LIN {X 0,Y 523.426,Z 552.768,A -85,B 0,C 180,E1 -4856.921,E2 -4856.921} C_VEL
LIN {X 0,Y 523.34,Z 554.167,A -85,B 0,C 180,E1 -4857.691,E2 -4857.691} C_VEL
LIN {X 0,Y 523.284,Z 555.786,A -85,B 0,C 180,E1 -4859.23,E2 -4859.23} C_VEL
LIN {X 0,Y 523.28,Z 556.011,A -85,B 0,C 180,E1 -4860,E2 -4860} C_VEL
LIN {X 0,Y 523.293,Z 555.206,A -85,B 0,C 180,E1 -4861.539,E2 -4861.539} C_VEL
LIN {X 0,Y 523.336,Z 554.266,A -85,B 0,C 180,E1 -4862.309,E2 -4862.309} C_VEL
LIN {X 0,Y 523.425,Z 552.886,A -85,B 0,C 180,E1 -4863.079,E2 -4863.079} C_VEL
LIN {X 0,Y 523.463,Z 550.021,A -85,B 0,C 180,E1 -4864.235,E2 -4864.235} C_VEL
LIN {X 0,Y 523.47,Z 546.108,A -85,B 0,C 180,E1 -4865.393,E2 -4865.393} C_VEL
LIN {X 0,Y 523.631,Z 540.404,A -85,B 0,C 180,E1 -4866.68,E2 -4866.68} C_VEL
LIN {X 0,Y 523.781,Z 533.513,A -85,B 0,C 180,E1 -4867.905,E2 -4867.905} C_VEL
LIN {X 0,Y 523.955,Z 525.259,A -85,B 0,C 180,E1 -4869.068,E2 -4869.068} C_VEL
LIN {X 0,Y 524.184,Z 516.803,A -85,B 0,C 180,E1 -4870.038,E2 -4870.038} C_VEL
LIN {X 0,Y 524.436,Z 506.403,A -85,B 0,C 180,E1 -4871.009,E2 -4871.009} C_VEL
LIN {X 0,Y 524.706,Z 495.922,A -85,B 0,C 180,E1 -4871.792,E2 -4871.792} C_VEL
LIN {X 0,Y 524.944,Z 484.563,A -85,B 0,C 180,E1 -4872.467,E2 -4872.467} C_VEL
LIN {X 0,Y 525.223,Z 471.548,A -85,B 0,C 180,E1 -4873.05,E2 -4873.05} C_VEL
LIN {X 0,Y 525.409,Z 458.329,A -85,B 0,C 180,E1 -4873.464,E2 -4873.464} C_VEL
LIN {X 0,Y 525.511,Z 443.709,A -85,B 0,C 180,E1 -4873.732,E2 -4873.732} C_VEL
LIN {X 0,Y 525.857,Z 355.697,A -85,B 0,C 180,E1 -4874.977,E2 -4874.977} C_VEL
LIN {X 0,Y 524.154,Z 347.018,A -85,B 0,C 180,E1 -4875.165,E2 -4875.165} C_VEL
LIN {X 0,Y 523.969,Z 341.219,A -85,B 0,C 180,E1 -4876.51,E2 -4876.51} C_VEL
LIN {X 0,Y 523.978,Z 341.218,A -85,B 0,C 180,E1 -4879.592,E2 -4879.592} C_VEL
LIN {X 0,Y 523.924,Z 341.219,A -85,B 0,C 180,E1 -4882.243,E2 -4882.243} C_VEL
LIN {X 0,Y 523.952,Z 341.222,A -85,B 0,C 180,E1 -4885.419,E2 -4885.419} C_VEL
LIN {X 0,Y 523.942,Z 341.217,A -85,B 0,C 180,E1 -4888.448,E2 -4888.448} C_VEL
LIN {X 0,Y 523.925,Z 341.223,A -85,B 0,C 180,E1 -4891.544,E2 -4891.544} C_VEL
LIN {X 0,Y 523.919,Z 341.221,A -85,B 0,C 180,E1 -4891.797,E2 -4891.797} C_VEL
LIN {X 0,Y 523.258,Z 341.303,A -85,B 0,C 180,E1 -4892.439,E2 -4892.439} C_VEL
LIN {X 0,Y 520.407,Z 341.662,A -85,B 0,C 180,E1 -4893.482,E2 -4893.482} C_VEL
LIN {X 0,Y 517.993,Z 341.962,A -85,B 0,C 180,E1 -4894.321,E2 -4894.321} C_VEL
LIN {X 0,Y 516.956,Z 342.094,A -85,B 0,C 180,E1 -4894.97,E2 -4894.97} C_VEL
LIN {X 0,Y 516.871,Z 342.103,A -85,B 0,C 180,E1 -4895.189,E2 -4895.189} C_VEL
LIN {X 0,Y 516.885,Z 342.097,A -85,B 0,C 180,E1 -4897.943,E2 -4897.943} C_VEL
LIN {X 0,Y 516.89,Z 342.1,A -85,B 0,C 180,E1 -4900.741,E2 -4900.741} C_VEL
LIN {X 0,Y 516.889,Z 342.101,A -85,B 0,C 180,E1 -4902.831,E2 -4902.831} C_VEL
LIN {X 0,Y 516.927,Z 342.097,A -85,B 0,C 180,E1 -4905.01,E2 -4905.01} C_VEL
LIN {X 0,Y 516.917,Z 342.094,A -85,B 0,C 180,E1 -4908.398,E2 -4908.398} C_VEL
LIN {X 0,Y 516.887,Z 342.1,A -85,B 0,C 180,E1 -4911.284,E2 -4911.284} C_VEL
LIN {X 0,Y 516.878,Z 342.098,A -85,B 0,C 180,E1 -4914.219,E2 -4914.219} C_VEL
LIN {X 0,Y 516.899,Z 342.1,A -85,B 0,C 180,E1 -4917.053,E2 -4917.053} C_VEL
LIN {X 0,Y 516.897,Z 342.095,A -85,B 0,C 180,E1 -4919.796,E2 -4919.796} C_VEL
LIN {X 0,Y 516.93,Z 342.094,A -85,B 0,C 180,E1 -4922.467,E2 -4922.467} C_VEL
LIN {X 0,Y 516.915,Z 342.097,A -85,B 0,C 180,E1 -4925.071,E2 -4925.071} C_VEL
LIN {X 0,Y 516.874,Z 342.098,A -85,B 0,C 180,E1 -4927.621,E2 -4927.621} C_VEL
LIN {X 0,Y 516.936,Z 342.091,A -85,B 0,C 180,E1 -4930.129,E2 -4930.129} C_VEL
LIN {X 0,Y 516.933,Z 342.097,A -85,B 0,C 180,E1 -4932.596,E2 -4932.596} C_VEL
LIN {X 0,Y 516.946,Z 342.093,A -85,B 0,C 180,E1 -4935.029,E2 -4935.029} C_VEL
LIN {X 0,Y 516.969,Z 342.088,A -85,B 0,C 180,E1 -4938.233,E2 -4938.233} C_VEL
LIN {X 0,Y 516.972,Z 342.086,A -85,B 0,C 180,E1 -4941.399,E2 -4941.399} C_VEL
LIN {X 0,Y 517.006,Z 342.081,A -85,B 0,C 180,E1 -4943.756,E2 -4943.756} C_VEL
LIN {X 0,Y 517.017,Z 342.084,A -85,B 0,C 180,E1 -4946.882,E2 -4946.882} C_VEL
LIN {X 0,Y 517.088,Z 342.073,A -85,B 0,C 180,E1 -4949.999,E2 -4949.999} C_VEL
LIN {X 0,Y 517.016,Z 342.081,A -85,B 0,C 180,E1 -4953.116,E2 -4953.116} C_VEL
LIN {X 0,Y 517.017,Z 342.085,A -85,B 0,C 180,E1 -4956.242,E2 -4956.242} C_VEL
LIN {X 0,Y 516.956,Z 342.087,A -85,B 0,C 180,E1 -4959.388,E2 -4959.388} C_VEL
LIN {X 0,Y 516.953,Z 342.089,A -85,B 0,C 180,E1 -4961.807,E2 -4961.807} C_VEL
LIN {X 0,Y 516.944,Z 342.089,A -85,B 0,C 180,E1 -4965.146,E2 -4965.146} C_VEL
LIN {X 0,Y 516.926,Z 342.098,A -85,B 0,C 180,E1 -4968.221,E2 -4968.221} C_VEL
LIN {X 0,Y 516.911,Z 342.096,A -85,B 0,C 180,E1 -4970.7,E2 -4970.7} C_VEL
LIN {X 0,Y 516.91,Z 342.099,A -85,B 0,C 180,E1 -4974.071,E2 -4974.071} C_VEL
LIN {X 0,Y 516.927,Z 342.093,A -85,B 0,C 180,E1 -4976.656,E2 -4976.656} C_VEL
LIN {X 0,Y 516.922,Z 342.092,A -85,B 0,C 180,E1 -4979.526,E2 -4979.526} C_VEL
LIN {X 0,Y 516.898,Z 342.098,A -85,B 0,C 180,E1 -4982.544,E2 -4982.544} C_VEL
LIN {X 0,Y 516.88,Z 342.096,A -85,B 0,C 180,E1 -4985.332,E2 -4985.332} C_VEL
LIN {X 0,Y 516.878,Z 342.103,A -85,B 0,C 180,E1 -4987.943,E2 -4987.943} C_VEL
LIN {X 0,Y 516.907,Z 342.094,A -85,B 0,C 180,E1 -4990.738,E2 -4990.738} C_VEL
LIN {X 0,Y 516.876,Z 342.103,A -85,B 0,C 180,E1 -4993.902,E2 -4993.902} C_VEL
LIN {X 0,Y 516.877,Z 342.103,A -85,B 0,C 180,E1 -4996.106,E2 -4996.106} C_VEL
LIN {X 0,Y 516.91,Z 342.093,A -85,B 0,C 180,E1 -4999.261,E2 -4999.261} C_VEL
LIN {X 0,Y 516.875,Z 342.103,A -85,B 0,C 180,E1 -5002.056,E2 -5002.056} C_VEL
LIN {X 0,Y 516.889,Z 342.095,A -85,B 0,C 180,E1 -5005.176,E2 -5005.176} C_VEL
LIN {X 0,Y 516.876,Z 342.103,A -85,B 0,C 180,E1 -5007.975,E2 -5007.975} C_VEL
LIN {X 0,Y 516.928,Z 342.09,A -85,B 0,C 180,E1 -5010.696,E2 -5010.696} C_VEL
LIN {X 0,Y 516.936,Z 342.097,A -85,B 0,C 180,E1 -5013.803,E2 -5013.803} C_VEL
LIN {X 0,Y 516.863,Z 342.098,A -85,B 0,C 180,E1 -5016.776,E2 -5016.776} C_VEL
LIN {X 0,Y 516.93,Z 342.098,A -85,B 0,C 180,E1 -5019.731,E2 -5019.731} C_VEL
LIN {X 0,Y 516.922,Z 342.09,A -85,B 0,C 180,E1 -5022.596,E2 -5022.596} C_VEL
LIN {X 0,Y 516.932,Z 342.09,A -85,B 0,C 180,E1 -5025.03,E2 -5025.03} C_VEL
LIN {X 0,Y 516.994,Z 342.083,A -85,B 0,C 180,E1 -5028.234,E2 -5028.234} C_VEL
LIN {X 0,Y 516.963,Z 342.091,A -85,B 0,C 180,E1 -5031.4,E2 -5031.4} C_VEL
LIN {X 0,Y 517.001,Z 342.086,A -85,B 0,C 180,E1 -5033.757,E2 -5033.757} C_VEL
LIN {X 0,Y 517.075,Z 342.078,A -85,B 0,C 180,E1 -5037.663,E2 -5037.663} C_VEL
LIN {X 0,Y 517.086,Z 342.07,A -85,B 0,C 180,E1 -5040.779,E2 -5040.779} C_VEL
LIN {X 0,Y 517.008,Z 342.083,A -85,B 0,C 180,E1 -5043.117,E2 -5043.117} C_VEL
LIN {X 0,Y 517.001,Z 342.08,A -85,B 0,C 180,E1 -5046.243,E2 -5046.243} C_VEL
LIN {X 0,Y 516.947,Z 342.095,A -85,B 0,C 180,E1 -5049.389,E2 -5049.389} C_VEL
LIN {X 0,Y 516.974,Z 342.086,A -85,B 0,C 180,E1 -5051.824,E2 -5051.824} C_VEL
LIN {X 0,Y 516.934,Z 342.094,A -85,B 0,C 180,E1 -5055.147,E2 -5055.147} C_VEL
LIN {X 0,Y 516.917,Z 342.091,A -85,B 0,C 180,E1 -5058.223,E2 -5058.223} C_VEL
LIN {X 0,Y 516.904,Z 342.094,A -85,B 0,C 180,E1 -5060.702,E2 -5060.702} C_VEL
LIN {X 0,Y 516.903,Z 342.093,A -85,B 0,C 180,E1 -5064.073,E2 -5064.073} C_VEL
LIN {X 0,Y 516.922,Z 342.092,A -85,B 0,C 180,E1 -5066.658,E2 -5066.658} C_VEL
LIN {X 0,Y 516.904,Z 342.097,A -85,B 0,C 180,E1 -5069.525,E2 -5069.525} C_VEL
LIN {X 0,Y 516.894,Z 342.095,A -85,B 0,C 180,E1 -5072.545,E2 -5072.545} C_VEL
LIN {X 0,Y 516.877,Z 342.102,A -85,B 0,C 180,E1 -5075.333,E2 -5075.333} C_VEL
LIN {X 0,Y 516.879,Z 342.096,A -85,B 0,C 180,E1 -5077.945,E2 -5077.945} C_VEL
LIN {X 0,Y 516.903,Z 342.097,A -85,B 0,C 180,E1 -5080.74,E2 -5080.74} C_VEL
LIN {X 0,Y 516.878,Z 342.096,A -85,B 0,C 180,E1 -5083.904,E2 -5083.904} C_VEL
LIN {X 0,Y 516.877,Z 342.096,A -85,B 0,C 180,E1 -5086.108,E2 -5086.108} C_VEL
LIN {X 0,Y 516.9,Z 342.098,A -85,B 0,C 180,E1 -5089.261,E2 -5089.261} C_VEL
LIN {X 0,Y 516.882,Z 342.096,A -85,B 0,C 180,E1 -5092.057,E2 -5092.057} C_VEL
LIN {X 0,Y 516.893,Z 342.099,A -85,B 0,C 180,E1 -5095.177,E2 -5095.177} C_VEL
LIN {X 0,Y 516.881,Z 342.096,A -85,B 0,C 180,E1 -5097.977,E2 -5097.977} C_VEL
LIN {X 0,Y 516.935,Z 342.098,A -85,B 0,C 180,E1 -5100.698,E2 -5100.698} C_VEL
LIN {X 0,Y 516.992,Z 342.265,A -85,B 0,C 180,E1 -5103.471,E2 -5103.471} C_VEL
LIN {X 0,Y 519.048,Z 353.214,A -85,B 0,C 180,E1 -5105.183,E2 -5105.183} C_VEL
LIN {X 0,Y 518.474,Z 372.179,A -85,B 0,C 180,E1 -5107.905,E2 -5107.905} C_VEL
LIN {X 0,Y 517.985,Z 392.732,A -85,B 0,C 180,E1 -5110.792,E2 -5110.792} C_VEL
LIN {X 0,Y 517.499,Z 414.528,A -85,B 0,C 180,E1 -5113.836,E2 -5113.836} C_VEL
LIN {X 0,Y 517.395,Z 420.236,A -85,B 0,C 180,E1 -5114.63,E2 -5114.63} C_VEL
LIN {X 0,Y 518.999,Z 433.665,A -85,B 0,C 180,E1 -5114.896,E2 -5114.896} C_VEL
LIN {X 0,Y 518.525,Z 525.57,A -85,B 0,C 180,E1 -5116.205,E2 -5116.205} C_VEL
LIN {X 0,Y 518.295,Z 538.806,A -85,B 0,C 180,E1 -5116.499,E2 -5116.499} C_VEL
LIN {X 0,Y 518.091,Z 550.95,A -85,B 0,C 180,E1 -5116.918,E2 -5116.918} C_VEL
LIN {X 0,Y 517.785,Z 563.865,A -85,B 0,C 180,E1 -5117.539,E2 -5117.539} C_VEL
LIN {X 0,Y 517.511,Z 575.181,A -85,B 0,C 180,E1 -5118.247,E2 -5118.247} C_VEL
LIN {X 0,Y 517.231,Z 586.403,A -85,B 0,C 180,E1 -5119.134,E2 -5119.134} C_VEL
LIN {X 0,Y 516.975,Z 595.488,A -85,B 0,C 180,E1 -5120.02,E2 -5120.02} C_VEL
LIN {X 0,Y 516.717,Z 605.338,A -85,B 0,C 180,E1 -5121.199,E2 -5121.199} C_VEL
LIN {X 0,Y 516.538,Z 613.202,A -85,B 0,C 180,E1 -5122.378,E2 -5122.378} C_VEL
LIN {X 0,Y 516.432,Z 618.939,A -85,B 0,C 180,E1 -5123.435,E2 -5123.435} C_VEL
LIN {X 0,Y 516.396,Z 623.777,A -85,B 0,C 180,E1 -5124.534,E2 -5124.534} C_VEL
LIN {X 0,Y 516.344,Z 627.812,A -85,B 0,C 180,E1 -5125.708,E2 -5125.708} C_VEL
LIN {X 0,Y 516.294,Z 630.787,A -85,B 0,C 180,E1 -5126.88,E2 -5126.88} C_VEL
LIN {X 0,Y 516.261,Z 632.203,A -85,B 0,C 180,E1 -5127.66,E2 -5127.66} C_VEL
LIN {X 0,Y 516.176,Z 633.82,A -85,B 0,C 180,E1 -5129.221,E2 -5129.221} C_VEL
LIN {X 0,Y 516.177,Z 634.032,A -85,B 0,C 180,E1 -5130.001,E2 -5130.001} C_VEL
LIN {X 0,Y 516.177,Z 633.806,A -85,B 0,C 180,E1 -5130.781,E2 -5130.781} C_VEL
LIN {X 0,Y 516.262,Z 632.169,A -85,B 0,C 180,E1 -5132.341,E2 -5132.341} C_VEL
LIN {X 0,Y 516.339,Z 630.735,A -85,B 0,C 180,E1 -5133.122,E2 -5133.122} C_VEL
LIN {X 0,Y 516.361,Z 627.727,A -85,B 0,C 180,E1 -5134.294,E2 -5134.294} C_VEL
LIN {X 0,Y 516.397,Z 623.654,A -85,B 0,C 180,E1 -5135.468,E2 -5135.468} C_VEL
LIN {X 0,Y 516.459,Z 617.536,A -85,B 0,C 180,E1 -5136.81,E2 -5136.81} C_VEL
LIN {X 0,Y 516.586,Z 610.535,A -85,B 0,C 180,E1 -5138.017,E2 -5138.017} C_VEL
LIN {X 0,Y 516.778,Z 602.01,A -85,B 0,C 180,E1 -5139.196,E2 -5139.196} C_VEL
LIN {X 0,Y 516.993,Z 593.236,A -85,B 0,C 180,E1 -5140.18,E2 -5140.18} C_VEL
LIN {X 0,Y 517.253,Z 582.419,A -85,B 0,C 180,E1 -5141.165,E2 -5141.165} C_VEL
LIN {X 0,Y 517.519,Z 571.704,A -85,B 0,C 180,E1 -5141.951,E2 -5141.951} C_VEL
LIN {X 0,Y 517.829,Z 559.727,A -85,B 0,C 180,E1 -5142.642,E2 -5142.642} C_VEL
LIN {X 0,Y 518.066,Z 547.312,A -85,B 0,C 180,E1 -5143.185,E2 -5143.185} C_VEL
LIN {X 0,Y 518.344,Z 533.734,A -85,B 0,C 180,E1 -5143.602,E2 -5143.602} C_VEL
LIN {X 0,Y 518.527,Z 518.504,A -85,B 0,C 180,E1 -5143.872,E2 -5143.872} C_VEL
LIN {X 0,Y 518.853,Z 431.421,A -85,B 0,C 180,E1 -5145.128,E2 -5145.128} C_VEL
LIN {X 0,Y 517.324,Z 419.204,A -85,B 0,C 180,E1 -5145.369,E2 -5145.369} C_VEL
LIN {X 0,Y 517.722,Z 395.583,A -85,B 0,C 180,E1 -5148.604,E2 -5148.604} C_VEL
LIN {X 0,Y 518.203,Z 373.38,A -85,B 0,C 180,E1 -5151.69,E2 -5151.69} C_VEL
LIN {X 0,Y 518.711,Z 352.398,A -85,B 0,C 180,E1 -5154.671,E2 -5154.671} C_VEL
LIN {X 0,Y 517.284,Z 343.864,A -85,B 0,C 180,E1 -5155.983,E2 -5155.983} C_VEL
LIN {X 0,Y 516.959,Z 342.092,A -85,B 0,C 180,E1 -5156.285,E2 -5156.285} C_VEL
LIN {X 0,Y 516.917,Z 342.098,A -85,B 0,C 180,E1 -5159.524,E2 -5159.524} C_VEL
LIN {X 0,Y 516.901,Z 342.097,A -85,B 0,C 180,E1 -5162.544,E2 -5162.544} C_VEL
LIN {X 0,Y 516.876,Z 342.104,A -85,B 0,C 180,E1 -5165.331,E2 -5165.331} C_VEL
LIN {X 0,Y 516.887,Z 342.097,A -85,B 0,C 180,E1 -5167.944,E2 -5167.944} C_VEL
LIN {X 0,Y 516.888,Z 342.101,A -85,B 0,C 180,E1 -5170.742,E2 -5170.742} C_VEL
LIN {X 0,Y 516.888,Z 342.101,A -85,B 0,C 180,E1 -5172.832,E2 -5172.832} C_VEL
LIN {X 0,Y 516.928,Z 342.097,A -85,B 0,C 180,E1 -5175.01,E2 -5175.01} C_VEL
LIN {X 0,Y 516.922,Z 342.092,A -85,B 0,C 180,E1 -5178.399,E2 -5178.399} C_VEL
LIN {X 0,Y 516.886,Z 342.1,A -85,B 0,C 180,E1 -5181.284,E2 -5181.284} C_VEL
LIN {X 0,Y 516.876,Z 342.097,A -85,B 0,C 180,E1 -5184.22,E2 -5184.22} C_VEL
LIN {X 0,Y 516.9,Z 342.101,A -85,B 0,C 180,E1 -5187.053,E2 -5187.053} C_VEL
LIN {X 0,Y 516.897,Z 342.095,A -85,B 0,C 180,E1 -5189.796,E2 -5189.796} C_VEL
LIN {X 0,Y 516.932,Z 342.094,A -85,B 0,C 180,E1 -5192.467,E2 -5192.467} C_VEL
LIN {X 0,Y 516.914,Z 342.099,A -85,B 0,C 180,E1 -5195.072,E2 -5195.072} C_VEL
LIN {X 0,Y 516.891,Z 342.102,A -85,B 0,C 180,E1 -5198.462,E2 -5198.462} C_VEL
LIN {X 0,Y 516.905,Z 342.1,A -85,B 0,C 180,E1 -5200.955,E2 -5200.955} C_VEL
LIN {X 0,Y 516.942,Z 342.242,A -85,B 0,C 180,E1 -5203.157,E2 -5203.157} C_VEL
LIN {X 0,Y 517.394,Z 346.715,A -85,B 0,C 180,E1 -5204.236,E2 -5204.236} C_VEL
LIN {X 0,Y 517.359,Z 348.857,A -85,B 0,C 180,E1 -5204.739,E2 -5204.739} C_VEL
LIN {X 0,Y 519.125,Z 357.781,A -85,B 0,C 180,E1 -5204.937,E2 -5204.937} C_VEL
LIN {X 0,Y 518.494,Z 454.508,A -85,B 0,C 180,E1 -5206.378,E2 -5206.378} C_VEL
LIN {X 0,Y 518.351,Z 468.183,A -85,B 0,C 180,E1 -5206.749,E2 -5206.749} C_VEL
LIN {X 0,Y 518.078,Z 481.002,A -85,B 0,C 180,E1 -5207.265,E2 -5207.265} C_VEL
LIN {X 0,Y 517.891,Z 492.363,A -85,B 0,C 180,E1 -5207.886,E2 -5207.886} C_VEL
LIN {X 0,Y 517.6,Z 503.312,A -85,B 0,C 180,E1 -5208.645,E2 -5208.645} C_VEL
LIN {X 0,Y 517.312,Z 513.559,A -85,B 0,C 180,E1 -5209.531,E2 -5209.531} C_VEL
LIN {X 0,Y 517.057,Z 523.54,A -85,B 0,C 180,E1 -5210.613,E2 -5210.613} C_VEL
LIN {X 0,Y 516.798,Z 532.275,A -85,B 0,C 180,E1 -5211.791,E2 -5211.791} C_VEL
LIN {X 0,Y 516.646,Z 539.255,A -85,B 0,C 180,E1 -5212.968,E2 -5212.968} C_VEL
LIN {X 0,Y 516.508,Z 544.792,A -85,B 0,C 180,E1 -5214.143,E2 -5214.143} C_VEL
LIN {X 0,Y 516.419,Z 549.131,A -85,B 0,C 180,E1 -5215.316,E2 -5215.316} C_VEL
LIN {X 0,Y 516.448,Z 551.434,A -85,B 0,C 180,E1 -5216.098,E2 -5216.098} C_VEL
LIN {X 0,Y 516.368,Z 553.298,A -85,B 0,C 180,E1 -5216.879,E2 -5216.879} C_VEL
LIN {X 0,Y 516.268,Z 554.716,A -85,B 0,C 180,E1 -5217.659,E2 -5217.659} C_VEL
LIN {X 0,Y 516.205,Z 556.324,A -85,B 0,C 180,E1 -5219.22,E2 -5219.22} C_VEL
LIN {X 0,Y 516.201,Z 556.545,A -85,B 0,C 180,E1 -5220,E2 -5220} C_VEL
LIN {X 0,Y 516.204,Z 556.349,A -85,B 0,C 180,E1 -5220.78,E2 -5220.78} C_VEL
LIN {X 0,Y 516.264,Z 554.775,A -85,B 0,C 180,E1 -5222.341,E2 -5222.341} C_VEL
LIN {X 0,Y 516.365,Z 553.39,A -85,B 0,C 180,E1 -5223.121,E2 -5223.121} C_VEL
LIN {X 0,Y 516.395,Z 550.503,A -85,B 0,C 180,E1 -5224.293,E2 -5224.293} C_VEL
LIN {X 0,Y 516.412,Z 546.576,A -85,B 0,C 180,E1 -5225.466,E2 -5225.466} C_VEL
LIN {X 0,Y 516.582,Z 541.168,A -85,B 0,C 180,E1 -5226.706,E2 -5226.706} C_VEL
LIN {X 0,Y 516.73,Z 535.121,A -85,B 0,C 180,E1 -5227.817,E2 -5227.817} C_VEL
LIN {X 0,Y 516.923,Z 527.127,A -85,B 0,C 180,E1 -5228.995,E2 -5228.995} C_VEL
LIN {X 0,Y 517.155,Z 518.946,A -85,B 0,C 180,E1 -5229.978,E2 -5229.978} C_VEL
LIN {X 0,Y 517.405,Z 508.952,A -85,B 0,C 180,E1 -5230.962,E2 -5230.962} C_VEL
LIN {X 0,Y 517.733,Z 497.741,A -85,B 0,C 180,E1 -5231.84,E2 -5231.84} C_VEL
LIN {X 0,Y 517.959,Z 486.48,A -85,B 0,C 180,E1 -5232.539,E2 -5232.539} C_VEL
LIN {X 0,Y 518.238,Z 474.069,A -85,B 0,C 180,E1 -5233.129,E2 -5233.129} C_VEL
LIN {X 0,Y 518.451,Z 460.807,A -85,B 0,C 180,E1 -5233.573,E2 -5233.573} C_VEL
LIN {X 0,Y 518.601,Z 447.927,A -85,B 0,C 180,E1 -5233.844,E2 -5233.844} C_VEL
LIN {X 0,Y 518.93,Z 356.14,A -85,B 0,C 180,E1 -5235.177,E2 -5235.177} C_VEL
LIN {X 0,Y 517.165,Z 347.479,A -85,B 0,C 180,E1 -5235.367,E2 -5235.367} C_VEL
LIN {X 0,Y 516.949,Z 342.094,A -85,B 0,C 180,E1 -5236.589,E2 -5236.589} C_VEL
LIN {X 0,Y 516.936,Z 342.092,A -85,B 0,C 180,E1 -5239.87,E2 -5239.87} C_VEL
LIN {X 0,Y 516.871,Z 342.098,A -85,B 0,C 180,E1 -5242.389,E2 -5242.389} C_VEL
LIN {X 0,Y 516.908,Z 342.097,A -85,B 0,C 180,E1 -5244.928,E2 -5244.928} C_VEL
LIN {X 0,Y 516.931,Z 342.095,A -85,B 0,C 180,E1 -5247.532,E2 -5247.532} C_VEL
LIN {X 0,Y 516.896,Z 342.095,A -85,B 0,C 180,E1 -5250.203,E2 -5250.203} C_VEL
LIN {X 0,Y 516.899,Z 342.1,A -85,B 0,C 180,E1 -5252.947,E2 -5252.947} C_VEL
LIN {X 0,Y 516.871,Z 342.103,A -85,B 0,C 180,E1 -5255.189,E2 -5255.189} C_VEL
LIN {X 0,Y 516.208,Z 342.187,A -85,B 0,C 180,E1 -5255.84,E2 -5255.84} C_VEL
LIN {X 0,Y 513.37,Z 342.54,A -85,B 0,C 180,E1 -5256.896,E2 -5256.896} C_VEL
LIN {X 0,Y 510.965,Z 342.836,A -85,B 0,C 180,E1 -5257.747,E2 -5257.747} C_VEL
LIN {X 0,Y 509.925,Z 342.964,A -85,B 0,C 180,E1 -5258.404,E2 -5258.404} C_VEL
LIN {X 0,Y 509.837,Z 342.974,A -85,B 0,C 180,E1 -5258.626,E2 -5258.626} C_VEL
LIN {X 0,Y 509.863,Z 342.971,A -85,B 0,C 180,E1 -5261.897,E2 -5261.897} C_VEL
LIN {X 0,Y 509.861,Z 342.976,A -85,B 0,C 180,E1 -5265.332,E2 -5265.332} C_VEL
LIN {X 0,Y 509.859,Z 342.975,A -85,B 0,C 180,E1 -5268.574,E2 -5268.574} C_VEL
LIN {X 0,Y 509.856,Z 342.972,A -85,B 0,C 180,E1 -5271.786,E2 -5271.786} C_VEL
LIN {X 0,Y 509.838,Z 342.979,A -85,B 0,C 180,E1 -5274.622,E2 -5274.622} C_VEL
LIN {X 0,Y 509.866,Z 342.972,A -85,B 0,C 180,E1 -5277.48,E2 -5277.48} C_VEL
LIN {X 0,Y 509.863,Z 342.973,A -85,B 0,C 180,E1 -5280.273,E2 -5280.273} C_VEL
LIN {X 0,Y 509.888,Z 342.973,A -85,B 0,C 180,E1 -5282.944,E2 -5282.944} C_VEL
LIN {X 0,Y 509.874,Z 342.97,A -85,B 0,C 180,E1 -5285.573,E2 -5285.573} C_VEL
LIN {X 0,Y 509.854,Z 342.977,A -85,B 0,C 180,E1 -5288.998,E2 -5288.998} C_VEL
LIN {X 0,Y 509.893,Z 342.968,A -85,B 0,C 180,E1 -5291.998,E2 -5291.998} C_VEL
LIN {X 0,Y 509.914,Z 342.97,A -85,B 0,C 180,E1 -5294.818,E2 -5294.818} C_VEL
LIN {X 0,Y 509.905,Z 342.968,A -85,B 0,C 180,E1 -5298.123,E2 -5298.123} C_VEL
LIN {X 0,Y 509.919,Z 342.965,A -85,B 0,C 180,E1 -5301.279,E2 -5301.279} C_VEL
LIN {X 0,Y 509.957,Z 342.959,A -85,B 0,C 180,E1 -5303.669,E2 -5303.669} C_VEL
LIN {X 0,Y 509.959,Z 342.963,A -85,B 0,C 180,E1 -5306.839,E2 -5306.839} C_VEL
LIN {X 0,Y 510.067,Z 342.946,A -85,B 0,C 180,E1 -5309.21,E2 -5309.21} C_VEL
LIN {X 0,Y 510.059,Z 342.953,A -85,B 0,C 180,E1 -5312.368,E2 -5312.368} C_VEL
LIN {X 0,Y 509.985,Z 342.962,A -85,B 0,C 180,E1 -5316.329,E2 -5316.329} C_VEL
LIN {X 0,Y 509.918,Z 342.968,A -85,B 0,C 180,E1 -5318.719,E2 -5318.719} C_VEL
LIN {X 0,Y 509.905,Z 342.968,A -85,B 0,C 180,E1 -5321.931,E2 -5321.931} C_VEL
LIN {X 0,Y 509.893,Z 342.967,A -85,B 0,C 180,E1 -5325.241,E2 -5325.241} C_VEL
LIN {X 0,Y 509.888,Z 342.971,A -85,B 0,C 180,E1 -5328,E2 -5328} C_VEL
LIN {X 0,Y 509.849,Z 342.973,A -85,B 0,C 180,E1 -5331.001,E2 -5331.001} C_VEL
LIN {X 0,Y 509.835,Z 342.975,A -85,B 0,C 180,E1 -5333.562,E2 -5333.562} C_VEL
LIN {X 0,Y 509.911,Z 342.97,A -85,B 0,C 180,E1 -5336.378,E2 -5336.378} C_VEL
LIN {X 0,Y 509.883,Z 342.969,A -85,B 0,C 180,E1 -5338.843,E2 -5338.843} C_VEL
LIN {X 0,Y 509.823,Z 342.977,A -85,B 0,C 180,E1 -5341.589,E2 -5341.589} C_VEL
LIN {X 0,Y 509.851,Z 342.976,A -85,B 0,C 180,E1 -5344.412,E2 -5344.412} C_VEL
LIN {X 0,Y 509.815,Z 342.977,A -85,B 0,C 180,E1 -5347.339,E2 -5347.339} C_VEL
LIN {X 0,Y 509.872,Z 342.973,A -85,B 0,C 180,E1 -5350.377,E2 -5350.377} C_VEL
LIN {X 0,Y 509.833,Z 342.974,A -85,B 0,C 180,E1 -5353.063,E2 -5353.063} C_VEL
LIN {X 0,Y 509.825,Z 342.98,A -85,B 0,C 180,E1 -5355.791,E2 -5355.791} C_VEL
LIN {X 0,Y 509.866,Z 342.971,A -85,B 0,C 180,E1 -5358.575,E2 -5358.575} C_VEL
LIN {X 0,Y 509.849,Z 342.978,A -85,B 0,C 180,E1 -5361.785,E2 -5361.785} C_VEL
LIN {X 0,Y 509.839,Z 342.974,A -85,B 0,C 180,E1 -5364.623,E2 -5364.623} C_VEL
LIN {X 0,Y 509.858,Z 342.974,A -85,B 0,C 180,E1 -5367.481,E2 -5367.481} C_VEL
LIN {X 0,Y 509.873,Z 342.972,A -85,B 0,C 180,E1 -5370.268,E2 -5370.268} C_VEL
LIN {X 0,Y 509.879,Z 342.968,A -85,B 0,C 180,E1 -5372.944,E2 -5372.944} C_VEL
LIN {X 0,Y 509.861,Z 342.976,A -85,B 0,C 180,E1 -5375.574,E2 -5375.574} C_VEL
LIN {X 0,Y 509.814,Z 342.979,A -85,B 0,C 180,E1 -5378.148,E2 -5378.148} C_VEL
LIN {X 0,Y 509.856,Z 342.97,A -85,B 0,C 180,E1 -5380.681,E2 -5380.681} C_VEL
LIN {X 0,Y 509.879,Z 342.97,A -85,B 0,C 180,E1 -5383.175,E2 -5383.175} C_VEL
LIN {X 0,Y 509.855,Z 342.979,A -85,B 0,C 180,E1 -5385.634,E2 -5385.634} C_VEL
LIN {X 0,Y 509.916,Z 342.963,A -85,B 0,C 180,E1 -5388.875,E2 -5388.875} C_VEL
LIN {X 0,Y 509.943,Z 342.962,A -85,B 0,C 180,E1 -5392.078,E2 -5392.078} C_VEL
LIN {X 0,Y 509.974,Z 342.955,A -85,B 0,C 180,E1 -5394.464,E2 -5394.464} C_VEL
LIN {X 0,Y 510.046,Z 342.954,A -85,B 0,C 180,E1 -5397.631,E2 -5397.631} C_VEL
LIN {X 0,Y 510.056,Z 342.946,A -85,B 0,C 180,E1 -5400.79,E2 -5400.79} C_VEL
LIN {X 0,Y 509.95,Z 342.962,A -85,B 0,C 180,E1 -5403.16,E2 -5403.16} C_VEL
LIN {X 0,Y 509.969,Z 342.956,A -85,B 0,C 180,E1 -5406.33,E2 -5406.33} C_VEL
LIN {X 0,Y 509.908,Z 342.964,A -85,B 0,C 180,E1 -5408.72,E2 -5408.72} C_VEL
LIN {X 0,Y 509.941,Z 342.961,A -85,B 0,C 180,E1 -5411.931,E2 -5411.931} C_VEL
LIN {X 0,Y 509.884,Z 342.974,A -85,B 0,C 180,E1 -5415.242,E2 -5415.242} C_VEL
LIN {X 0,Y 509.88,Z 342.968,A -85,B 0,C 180,E1 -5418.002,E2 -5418.002} C_VEL
LIN {X 0,Y 509.842,Z 342.976,A -85,B 0,C 180,E1 -5421.002,E2 -5421.002} C_VEL
LIN {X 0,Y 509.828,Z 342.978,A -85,B 0,C 180,E1 -5423.564,E2 -5423.564} C_VEL
LIN {X 0,Y 509.906,Z 342.964,A -85,B 0,C 180,E1 -5426.38,E2 -5426.38} C_VEL
LIN {X 0,Y 509.87,Z 342.972,A -85,B 0,C 180,E1 -5428.845,E2 -5428.845} C_VEL
LIN {X 0,Y 509.818,Z 342.978,A -85,B 0,C 180,E1 -5431.59,E2 -5431.59} C_VEL
LIN {X 0,Y 509.848,Z 342.972,A -85,B 0,C 180,E1 -5434.414,E2 -5434.414} C_VEL
LIN {X 0,Y 509.816,Z 342.981,A -85,B 0,C 180,E1 -5437.341,E2 -5437.341} C_VEL
LIN {X 0,Y 509.857,Z 342.971,A -85,B 0,C 180,E1 -5440.381,E2 -5440.381} C_VEL
LIN {X 0,Y 509.836,Z 342.981,A -85,B 0,C 180,E1 -5443.065,E2 -5443.065} C_VEL
LIN {X 0,Y 509.825,Z 342.975,A -85,B 0,C 180,E1 -5445.793,E2 -5445.793} C_VEL
LIN {X 0,Y 509.861,Z 342.973,A -85,B 0,C 180,E1 -5448.577,E2 -5448.577} C_VEL
LIN {X 0,Y 509.854,Z 342.971,A -85,B 0,C 180,E1 -5451.786,E2 -5451.786} C_VEL
LIN {X 0,Y 509.844,Z 342.977,A -85,B 0,C 180,E1 -5454.624,E2 -5454.624} C_VEL
LIN {X 0,Y 509.863,Z 342.972,A -85,B 0,C 180,E1 -5457.482,E2 -5457.482} C_VEL
LIN {X 0,Y 509.88,Z 342.972,A -85,B 0,C 180,E1 -5460.27,E2 -5460.27} C_VEL
LIN {X 0,Y 509.926,Z 343.084,A -85,B 0,C 180,E1 -5463.256,E2 -5463.256} C_VEL
LIN {X 0,Y 512.141,Z 354.531,A -85,B 0,C 180,E1 -5465.072,E2 -5465.072} C_VEL
LIN {X 0,Y 511.533,Z 373.256,A -85,B 0,C 180,E1 -5467.802,E2 -5467.802} C_VEL
LIN {X 0,Y 510.996,Z 393.762,A -85,B 0,C 180,E1 -5470.727,E2 -5470.727} C_VEL
LIN {X 0,Y 510.475,Z 415.528,A -85,B 0,C 180,E1 -5473.813,E2 -5473.813} C_VEL
LIN {X 0,Y 510.381,Z 420.011,A -85,B 0,C 180,E1 -5474.429,E2 -5474.429} C_VEL
LIN {X 0,Y 512.138,Z 433.769,A -85,B 0,C 180,E1 -5474.698,E2 -5474.698} C_VEL
LIN {X 0,Y 511.588,Z 525.536,A -85,B 0,C 180,E1 -5476.04,E2 -5476.04} C_VEL
LIN {X 0,Y 511.331,Z 539.44,A -85,B 0,C 180,E1 -5476.362,E2 -5476.362} C_VEL
LIN {X 0,Y 511.046,Z 552.316,A -85,B 0,C 180,E1 -5476.835,E2 -5476.835} C_VEL
LIN {X 0,Y 510.764,Z 564.614,A -85,B 0,C 180,E1 -5477.455,E2 -5477.455} C_VEL
LIN {X 0,Y 510.468,Z 575.839,A -85,B 0,C 180,E1 -5478.184,E2 -5478.184} C_VEL
LIN {X 0,Y 510.174,Z 586.789,A -85,B 0,C 180,E1 -5479.082,E2 -5479.082} C_VEL
LIN {X 0,Y 509.873,Z 596.635,A -85,B 0,C 180,E1 -5480.08,E2 -5480.08} C_VEL
LIN {X 0,Y 509.664,Z 604.711,A -85,B 0,C 180,E1 -5481.077,E2 -5481.077} C_VEL
LIN {X 0,Y 509.445,Z 612.61,A -85,B 0,C 180,E1 -5482.271,E2 -5482.271} C_VEL
LIN {X 0,Y 509.349,Z 618.835,A -85,B 0,C 180,E1 -5483.444,E2 -5483.444} C_VEL
LIN {X 0,Y 509.246,Z 624.672,A -85,B 0,C 180,E1 -5484.854,E2 -5484.854} C_VEL
LIN {X 0,Y 509.3,Z 628.362,A -85,B 0,C 180,E1 -5486.045,E2 -5486.045} C_VEL
LIN {X 0,Y 509.212,Z 630.255,A -85,B 0,C 180,E1 -5486.836,E2 -5486.836} C_VEL
LIN {X 0,Y 509.19,Z 631.677,A -85,B 0,C 180,E1 -5487.628,E2 -5487.628} C_VEL
LIN {X 0,Y 509.095,Z 633.293,A -85,B 0,C 180,E1 -5489.21,E2 -5489.21} C_VEL
LIN {X 0,Y 509.097,Z 633.504,A -85,B 0,C 180,E1 -5490.001,E2 -5490.001} C_VEL
LIN {X 0,Y 509.096,Z 633.273,A -85,B 0,C 180,E1 -5490.792,E2 -5490.792} C_VEL
LIN {X 0,Y 509.193,Z 631.618,A -85,B 0,C 180,E1 -5492.374,E2 -5492.374} C_VEL
LIN {X 0,Y 509.253,Z 630.171,A -85,B 0,C 180,E1 -5493.165,E2 -5493.165} C_VEL
LIN {X 0,Y 509.266,Z 627.141,A -85,B 0,C 180,E1 -5494.354,E2 -5494.354} C_VEL
LIN {X 0,Y 509.331,Z 623.043,A -85,B 0,C 180,E1 -5495.544,E2 -5495.544} C_VEL
LIN {X 0,Y 509.381,Z 617.146,A -85,B 0,C 180,E1 -5496.855,E2 -5496.855} C_VEL
LIN {X 0,Y 509.504,Z 609.835,A -85,B 0,C 180,E1 -5498.129,E2 -5498.129} C_VEL
LIN {X 0,Y 509.721,Z 601.259,A -85,B 0,C 180,E1 -5499.324,E2 -5499.324} C_VEL
LIN {X 0,Y 509.957,Z 591.429,A -85,B 0,C 180,E1 -5500.422,E2 -5500.422} C_VEL
LIN {X 0,Y 510.262,Z 580.323,A -85,B 0,C 180,E1 -5501.42,E2 -5501.42} C_VEL
LIN {X 0,Y 510.497,Z 569.647,A -85,B 0,C 180,E1 -5502.188,E2 -5502.188} C_VEL
LIN {X 0,Y 510.853,Z 557.603,A -85,B 0,C 180,E1 -5502.868,E2 -5502.868} C_VEL
LIN {X 0,Y 511.129,Z 544.73,A -85,B 0,C 180,E1 -5503.417,E2 -5503.417} C_VEL
LIN {X 0,Y 511.417,Z 532.02,A -85,B 0,C 180,E1 -5503.789,E2 -5503.789} C_VEL
LIN {X 0,Y 511.655,Z 512.836,A -85,B 0,C 180,E1 -5504.112,E2 -5504.112} C_VEL
LIN {X 0,Y 512.032,Z 432.599,A -85,B 0,C 180,E1 -5505.305,E2 -5505.305} C_VEL
LIN {X 0,Y 510.276,Z 418.563,A -85,B 0,C 180,E1 -5505.579,E2 -5505.579} C_VEL
LIN {X 0,Y 510.761,Z 394.947,A -85,B 0,C 180,E1 -5508.867,E2 -5508.867} C_VEL
LIN {X 0,Y 511.331,Z 371.344,A -85,B 0,C 180,E1 -5512.209,E2 -5512.209} C_VEL
LIN {X 0,Y 511.8,Z 354.312,A -85,B 0,C 180,E1 -5514.677,E2 -5514.677} C_VEL
LIN {X 0,Y 510.877,Z 347.866,A -85,B 0,C 180,E1 -5515.68,E2 -5515.68} C_VEL
LIN {X 0,Y 509.915,Z 342.971,A -85,B 0,C 180,E1 -5516.487,E2 -5516.487} C_VEL
LIN {X 0,Y 509.882,Z 342.975,A -85,B 0,C 180,E1 -5518.845,E2 -5518.845} C_VEL
LIN {X 0,Y 509.826,Z 342.98,A -85,B 0,C 180,E1 -5521.591,E2 -5521.591} C_VEL
LIN {X 0,Y 509.856,Z 342.974,A -85,B 0,C 180,E1 -5524.414,E2 -5524.414} C_VEL
LIN {X 0,Y 509.822,Z 342.982,A -85,B 0,C 180,E1 -5527.341,E2 -5527.341} C_VEL
LIN {X 0,Y 509.843,Z 342.975,A -85,B 0,C 180,E1 -5530.383,E2 -5530.383} C_VEL
LIN {X 0,Y 509.828,Z 342.982,A -85,B 0,C 180,E1 -5533.062,E2 -5533.062} C_VEL
LIN {X 0,Y 509.836,Z 342.975,A -85,B 0,C 180,E1 -5535.793,E2 -5535.793} C_VEL
LIN {X 0,Y 509.863,Z 342.973,A -85,B 0,C 180,E1 -5538.575,E2 -5538.575} C_VEL
LIN {X 0,Y 509.856,Z 342.972,A -85,B 0,C 180,E1 -5541.787,E2 -5541.787} C_VEL
LIN {X 0,Y 509.835,Z 342.978,A -85,B 0,C 180,E1 -5544.622,E2 -5544.622} C_VEL
LIN {X 0,Y 509.866,Z 342.972,A -85,B 0,C 180,E1 -5547.481,E2 -5547.481} C_VEL
LIN {X 0,Y 509.864,Z 342.973,A -85,B 0,C 180,E1 -5550.274,E2 -5550.274} C_VEL
LIN {X 0,Y 509.889,Z 342.974,A -85,B 0,C 180,E1 -5552.944,E2 -5552.944} C_VEL
LIN {X 0,Y 509.87,Z 342.972,A -85,B 0,C 180,E1 -5555.574,E2 -5555.574} C_VEL
LIN {X 0,Y 509.856,Z 342.979,A -85,B 0,C 180,E1 -5558.998,E2 -5558.998} C_VEL
LIN {X 0,Y 509.866,Z 342.975,A -85,B 0,C 180,E1 -5561.516,E2 -5561.516} C_VEL
LIN {X 0,Y 509.916,Z 343.125,A -85,B 0,C 180,E1 -5562.969,E2 -5562.969} C_VEL
LIN {X 0,Y 510.445,Z 348.844,A -85,B 0,C 180,E1 -5564.366,E2 -5564.366} C_VEL
LIN {X 0,Y 510.431,Z 349.664,A -85,B 0,C 180,E1 -5564.541,E2 -5564.541} C_VEL
LIN {X 0,Y 512.214,Z 357.707,A -85,B 0,C 180,E1 -5564.725,E2 -5564.725} C_VEL
LIN {X 0,Y 511.566,Z 455.115,A -85,B 0,C 180,E1 -5566.215,E2 -5566.215} C_VEL
LIN {X 0,Y 511.413,Z 468.761,A -85,B 0,C 180,E1 -5566.591,E2 -5566.591} C_VEL
LIN {X 0,Y 511.154,Z 481.08,A -85,B 0,C 180,E1 -5567.09,E2 -5567.09} C_VEL
LIN {X 0,Y 510.942,Z 493.233,A -85,B 0,C 180,E1 -5567.762,E2 -5567.762} C_VEL
LIN {X 0,Y 510.607,Z 504.871,A -85,B 0,C 180,E1 -5568.588,E2 -5568.588} C_VEL
LIN {X 0,Y 510.31,Z 514.906,A -85,B 0,C 180,E1 -5569.486,E2 -5569.486} C_VEL
LIN {X 0,Y 510.078,Z 523.942,A -85,B 0,C 180,E1 -5570.483,E2 -5570.483} C_VEL
LIN {X 0,Y 509.778,Z 532.73,A -85,B 0,C 180,E1 -5571.677,E2 -5571.677} C_VEL
LIN {X 0,Y 509.604,Z 539.736,A -85,B 0,C 180,E1 -5572.87,E2 -5572.87} C_VEL
LIN {X 0,Y 509.454,Z 545.302,A -85,B 0,C 180,E1 -5574.061,E2 -5574.061} C_VEL
LIN {X 0,Y 509.378,Z 549.66,A -85,B 0,C 180,E1 -5575.251,E2 -5575.251} C_VEL
LIN {X 0,Y 509.377,Z 551.957,A -85,B 0,C 180,E1 -5576.044,E2 -5576.044} C_VEL
LIN {X 0,Y 509.312,Z 553.827,A -85,B 0,C 180,E1 -5576.836,E2 -5576.836} C_VEL
LIN {X 0,Y 509.199,Z 555.254,A -85,B 0,C 180,E1 -5577.627,E2 -5577.627} C_VEL
LIN {X 0,Y 509.126,Z 556.857,A -85,B 0,C 180,E1 -5579.209,E2 -5579.209} C_VEL
LIN {X 0,Y 509.122,Z 557.079,A -85,B 0,C 180,E1 -5580,E2 -5580} C_VEL
LIN {X 0,Y 509.125,Z 556.884,A -85,B 0,C 180,E1 -5580.791,E2 -5580.791} C_VEL
LIN {X 0,Y 509.196,Z 555.284,A -85,B 0,C 180,E1 -5582.373,E2 -5582.373} C_VEL
LIN {X 0,Y 509.306,Z 553.893,A -85,B 0,C 180,E1 -5583.164,E2 -5583.164} C_VEL
LIN {X 0,Y 509.333,Z 550.984,A -85,B 0,C 180,E1 -5584.352,E2 -5584.352} C_VEL
LIN {X 0,Y 509.356,Z 547.04,A -85,B 0,C 180,E1 -5585.542,E2 -5585.542} C_VEL
LIN {X 0,Y 509.533,Z 541.936,A -85,B 0,C 180,E1 -5586.732,E2 -5586.732} C_VEL
LIN {X 0,Y 509.694,Z 535.515,A -85,B 0,C 180,E1 -5587.926,E2 -5587.926} C_VEL
LIN {X 0,Y 509.922,Z 527.478,A -85,B 0,C 180,E1 -5589.12,E2 -5589.12} C_VEL
LIN {X 0,Y 510.169,Z 519.264,A -85,B 0,C 180,E1 -5590.116,E2 -5590.116} C_VEL
LIN {X 0,Y 510.448,Z 509.22,A -85,B 0,C 180,E1 -5591.114,E2 -5591.114} C_VEL
LIN {X 0,Y 510.766,Z 498.226,A -85,B 0,C 180,E1 -5591.982,E2 -5591.982} C_VEL
LIN {X 0,Y 511.036,Z 486.604,A -85,B 0,C 180,E1 -5592.711,E2 -5592.711} C_VEL
LIN {X 0,Y 511.294,Z 475.252,A -85,B 0,C 180,E1 -5593.26,E2 -5593.26} C_VEL
LIN {X 0,Y 511.518,Z 462.349,A -85,B 0,C 180,E1 -5593.71,E2 -5593.71} C_VEL
LIN {X 0,Y 511.7,Z 448.742,A -85,B 0,C 180,E1 -5594.009,E2 -5594.009} C_VEL
LIN {X 0,Y 512.104,Z 357.086,A -85,B 0,C 180,E1 -5595.375,E2 -5595.375} C_VEL
LIN {X 0,Y 510.187,Z 347.85,A -85,B 0,C 180,E1 -5595.582,E2 -5595.582} C_VEL
LIN {X 0,Y 509.897,Z 342.973,A -85,B 0,C 180,E1 -5596.722,E2 -5596.722} C_VEL
LIN {X 0,Y 509.921,Z 342.964,A -85,B 0,C 180,E1 -5600.155,E2 -5600.155} C_VEL
LIN {X 0,Y 509.828,Z 342.98,A -85,B 0,C 180,E1 -5603.564,E2 -5603.564} C_VEL
LIN {X 0,Y 509.916,Z 342.965,A -85,B 0,C 180,E1 -5606.378,E2 -5606.378} C_VEL
LIN {X 0,Y 509.881,Z 342.973,A -85,B 0,C 180,E1 -5608.844,E2 -5608.844} C_VEL
LIN {X 0,Y 509.825,Z 342.979,A -85,B 0,C 180,E1 -5611.59,E2 -5611.59} C_VEL
LIN {X 0,Y 509.852,Z 342.973,A -85,B 0,C 180,E1 -5614.413,E2 -5614.413} C_VEL
LIN {X 0,Y 509.821,Z 342.981,A -85,B 0,C 180,E1 -5617.34,E2 -5617.34} C_VEL
LIN {X 0,Y 509.837,Z 342.974,A -85,B 0,C 180,E1 -5618.626,E2 -5618.626} C_VEL
LIN {X 0,Y 509.154,Z 343.064,A -85,B 0,C 180,E1 -5619.286,E2 -5619.286} C_VEL
LIN {X 0,Y 506.283,Z 343.418,A -85,B 0,C 180,E1 -5620.356,E2 -5620.356} C_VEL
LIN {X 0,Y 503.878,Z 343.721,A -85,B 0,C 180,E1 -5621.219,E2 -5621.219} C_VEL
LIN {X 0,Y 502.87,Z 343.843,A -85,B 0,C 180,E1 -5621.885,E2 -5621.885} C_VEL
LIN {X 0,Y 502.8,Z 343.851,A -85,B 0,C 180,E1 -5622.11,E2 -5622.11} C_VEL
LIN {X 0,Y 502.805,Z 343.853,A -85,B 0,C 180,E1 -5625.468,E2 -5625.468} C_VEL
LIN {X 0,Y 502.824,Z 343.853,A -85,B 0,C 180,E1 -5628.934,E2 -5628.934} C_VEL
LIN {X 0,Y 502.798,Z 343.851,A -85,B 0,C 180,E1 -5632.046,E2 -5632.046} C_VEL
LIN {X 0,Y 502.806,Z 343.855,A -85,B 0,C 180,E1 -5635.034,E2 -5635.034} C_VEL
LIN {X 0,Y 502.788,Z 343.853,A -85,B 0,C 180,E1 -5637.915,E2 -5637.915} C_VEL
LIN {X 0,Y 502.828,Z 343.854,A -85,B 0,C 180,E1 -5640.712,E2 -5640.712} C_VEL
LIN {X 0,Y 502.867,Z 343.844,A -85,B 0,C 180,E1 -5643.439,E2 -5643.439} C_VEL
LIN {X 0,Y 502.796,Z 343.852,A -85,B 0,C 180,E1 -5646.086,E2 -5646.086} C_VEL
LIN {X 0,Y 502.787,Z 343.858,A -85,B 0,C 180,E1 -5648.688,E2 -5648.688} C_VEL
LIN {X 0,Y 502.834,Z 343.849,A -85,B 0,C 180,E1 -5651.248,E2 -5651.248} C_VEL
LIN {X 0,Y 502.826,Z 343.848,A -85,B 0,C 180,E1 -5653.766,E2 -5653.766} C_VEL
LIN {X 0,Y 502.835,Z 343.849,A -85,B 0,C 180,E1 -5656.254,E2 -5656.254} C_VEL
LIN {X 0,Y 502.881,Z 343.846,A -85,B 0,C 180,E1 -5658.716,E2 -5658.716} C_VEL
LIN {X 0,Y 502.905,Z 343.839,A -85,B 0,C 180,E1 -5661.966,E2 -5661.966} C_VEL
LIN {X 0,Y 502.937,Z 343.839,A -85,B 0,C 180,E1 -5664.386,E2 -5664.386} C_VEL
LIN {X 0,Y 503.028,Z 343.822,A -85,B 0,C 180,E1 -5667.597,E2 -5667.597} C_VEL
LIN {X 0,Y 503.03,Z 343.824,A -85,B 0,C 180,E1 -5669.999,E2 -5669.999} C_VEL
LIN {X 0,Y 503.028,Z 343.829,A -85,B 0,C 180,E1 -5672.401,E2 -5672.401} C_VEL
LIN {X 0,Y 502.944,Z 343.833,A -85,B 0,C 180,E1 -5675.612,E2 -5675.612} C_VEL
LIN {X 0,Y 502.903,Z 343.841,A -85,B 0,C 180,E1 -5678.032,E2 -5678.032} C_VEL
LIN {X 0,Y 502.878,Z 343.841,A -85,B 0,C 180,E1 -5681.282,E2 -5681.282} C_VEL
LIN {X 0,Y 502.845,Z 343.849,A -85,B 0,C 180,E1 -5684.57,E2 -5684.57} C_VEL
LIN {X 0,Y 502.862,Z 343.846,A -85,B 0,C 180,E1 -5687.906,E2 -5687.906} C_VEL
LIN {X 0,Y 502.827,Z 343.851,A -85,B 0,C 180,E1 -5690.535,E2 -5690.535} C_VEL
LIN {X 0,Y 502.795,Z 343.851,A -85,B 0,C 180,E1 -5693.039,E2 -5693.039} C_VEL
LIN {X 0,Y 502.84,Z 343.847,A -85,B 0,C 180,E1 -5695.674,E2 -5695.674} C_VEL
LIN {X 0,Y 502.84,Z 343.85,A -85,B 0,C 180,E1 -5698.371,E2 -5698.371} C_VEL
LIN {X 0,Y 502.794,Z 343.852,A -85,B 0,C 180,E1 -5701.499,E2 -5701.499} C_VEL
LIN {X 0,Y 502.804,Z 343.854,A -85,B 0,C 180,E1 -5704.444,E2 -5704.444} C_VEL
LIN {X 0,Y 502.777,Z 343.853,A -85,B 0,C 180,E1 -5707.177,E2 -5707.177} C_VEL
LIN {X 0,Y 502.829,Z 343.854,A -85,B 0,C 180,E1 -5710.01,E2 -5710.01} C_VEL
LIN {X 0,Y 502.817,Z 343.853,A -85,B 0,C 180,E1 -5712.201,E2 -5712.201} C_VEL
LIN {X 0,Y 502.795,Z 343.852,A -85,B 0,C 180,E1 -5715.467,E2 -5715.467} C_VEL
LIN {X 0,Y 502.833,Z 343.853,A -85,B 0,C 180,E1 -5717.864,E2 -5717.864} C_VEL
LIN {X 0,Y 502.814,Z 343.848,A -85,B 0,C 180,E1 -5721.025,E2 -5721.025} C_VEL
LIN {X 0,Y 502.778,Z 343.857,A -85,B 0,C 180,E1 -5724.166,E2 -5724.166} C_VEL
LIN {X 0,Y 502.825,Z 343.847,A -85,B 0,C 180,E1 -5726.992,E2 -5726.992} C_VEL
LIN {X 0,Y 502.822,Z 343.852,A -85,B 0,C 180,E1 -5730.061,E2 -5730.061} C_VEL
LIN {X 0,Y 502.827,Z 343.847,A -85,B 0,C 180,E1 -5732.533,E2 -5732.533} C_VEL
LIN {X 0,Y 502.82,Z 343.849,A -85,B 0,C 180,E1 -5735.298,E2 -5735.298} C_VEL
LIN {X 0,Y 502.776,Z 343.86,A -85,B 0,C 180,E1 -5737.826,E2 -5737.826} C_VEL
LIN {X 0,Y 502.817,Z 343.848,A -85,B 0,C 180,E1 -5740.4,E2 -5740.4} C_VEL
LIN {X 0,Y 502.827,Z 343.846,A -85,B 0,C 180,E1 -5742.931,E2 -5742.931} C_VEL
LIN {X 0,Y 502.836,Z 343.85,A -85,B 0,C 180,E1 -5745.429,E2 -5745.429} C_VEL
LIN {X 0,Y 502.885,Z 343.839,A -85,B 0,C 180,E1 -5748.717,E2 -5748.717} C_VEL
LIN {X 0,Y 502.893,Z 343.841,A -85,B 0,C 180,E1 -5751.967,E2 -5751.967} C_VEL
LIN {X 0,Y 502.93,Z 343.833,A -85,B 0,C 180,E1 -5754.386,E2 -5754.386} C_VEL
LIN {X 0,Y 503.016,Z 343.83,A -85,B 0,C 180,E1 -5757.598,E2 -5757.598} C_VEL
LIN {X 0,Y 503.017,Z 343.824,A -85,B 0,C 180,E1 -5760,E2 -5760} C_VEL
LIN {X 0,Y 503.016,Z 343.822,A -85,B 0,C 180,E1 -5762.402,E2 -5762.402} C_VEL
LIN {X 0,Y 502.95,Z 343.837,A -85,B 0,C 180,E1 -5765.613,E2 -5765.613} C_VEL
LIN {X 0,Y 502.892,Z 343.839,A -85,B 0,C 180,E1 -5768.034,E2 -5768.034} C_VEL
LIN {X 0,Y 502.885,Z 343.845,A -85,B 0,C 180,E1 -5771.283,E2 -5771.283} C_VEL
LIN {X 0,Y 502.836,Z 343.845,A -85,B 0,C 180,E1 -5774.571,E2 -5774.571} C_VEL
LIN {X 0,Y 502.853,Z 343.844,A -85,B 0,C 180,E1 -5777.907,E2 -5777.907} C_VEL
LIN {X 0,Y 502.82,Z 343.847,A -85,B 0,C 180,E1 -5780.537,E2 -5780.537} C_VEL
LIN {X 0,Y 502.788,Z 343.856,A -85,B 0,C 180,E1 -5783.041,E2 -5783.041} C_VEL
LIN {X 0,Y 502.833,Z 343.848,A -85,B 0,C 180,E1 -5785.676,E2 -5785.676} C_VEL
LIN {X 0,Y 502.833,Z 343.846,A -85,B 0,C 180,E1 -5788.373,E2 -5788.373} C_VEL
LIN {X 0,Y 502.789,Z 343.855,A -85,B 0,C 180,E1 -5791.5,E2 -5791.5} C_VEL
LIN {X 0,Y 502.8,Z 343.85,A -85,B 0,C 180,E1 -5794.446,E2 -5794.446} C_VEL
LIN {X 0,Y 502.777,Z 343.861,A -85,B 0,C 180,E1 -5797.18,E2 -5797.18} C_VEL
LIN {X 0,Y 502.821,Z 343.847,A -85,B 0,C 180,E1 -5800.012,E2 -5800.012} C_VEL
LIN {X 0,Y 502.821,Z 343.847,A -85,B 0,C 180,E1 -5802.203,E2 -5802.203} C_VEL
LIN {X 0,Y 502.795,Z 343.853,A -85,B 0,C 180,E1 -5805.469,E2 -5805.469} C_VEL
LIN {X 0,Y 502.825,Z 343.847,A -85,B 0,C 180,E1 -5807.865,E2 -5807.865} C_VEL
LIN {X 0,Y 502.818,Z 343.856,A -85,B 0,C 180,E1 -5811.027,E2 -5811.027} C_VEL
LIN {X 0,Y 502.783,Z 343.853,A -85,B 0,C 180,E1 -5814.168,E2 -5814.168} C_VEL
LIN {X 0,Y 502.83,Z 343.854,A -85,B 0,C 180,E1 -5816.994,E2 -5816.994} C_VEL
LIN {X 0,Y 502.829,Z 343.85,A -85,B 0,C 180,E1 -5820.063,E2 -5820.063} C_VEL
LIN {X 0,Y 502.895,Z 343.959,A -85,B 0,C 180,E1 -5823.051,E2 -5823.051} C_VEL
LIN {X 0,Y 505.053,Z 354.512,A -85,B 0,C 180,E1 -5824.756,E2 -5824.756} C_VEL
LIN {X 0,Y 505.085,Z 361.235,A -85,B 0,C 180,E1 -5825.766,E2 -5825.766} C_VEL
LIN {X 0,Y 504.422,Z 381.661,A -85,B 0,C 180,E1 -5828.763,E2 -5828.763} C_VEL
LIN {X 0,Y 503.74,Z 404.929,A -85,B 0,C 180,E1 -5832.126,E2 -5832.126} C_VEL
LIN {X 0,Y 503.36,Z 419.422,A -85,B 0,C 180,E1 -5834.202,E2 -5834.202} C_VEL
LIN {X 0,Y 505.26,Z 434.407,A -85,B 0,C 180,E1 -5834.502,E2 -5834.502} C_VEL
LIN {X 0,Y 504.675,Z 526.918,A -85,B 0,C 180,E1 -5835.896,E2 -5835.896} C_VEL
LIN {X 0,Y 504.376,Z 539.95,A -85,B 0,C 180,E1 -5836.222,E2 -5836.222} C_VEL
LIN {X 0,Y 504.006,Z 553.655,A -85,B 0,C 180,E1 -5836.751,E2 -5836.751} C_VEL
LIN {X 0,Y 503.722,Z 566.248,A -85,B 0,C 180,E1 -5837.424,E2 -5837.424} C_VEL
LIN {X 0,Y 503.425,Z 576.413,A -85,B 0,C 180,E1 -5838.118,E2 -5838.118} C_VEL
LIN {X 0,Y 503.118,Z 587.177,A -85,B 0,C 180,E1 -5839.029,E2 -5839.029} C_VEL
LIN {X 0,Y 502.825,Z 595.976,A -85,B 0,C 180,E1 -5839.939,E2 -5839.939} C_VEL
LIN {X 0,Y 502.584,Z 604.082,A -85,B 0,C 180,E1 -5840.95,E2 -5840.95} C_VEL
LIN {X 0,Y 502.378,Z 612.02,A -85,B 0,C 180,E1 -5842.162,E2 -5842.162} C_VEL
LIN {X 0,Y 502.276,Z 618.681,A -85,B 0,C 180,E1 -5843.442,E2 -5843.442} C_VEL
LIN {X 0,Y 502.182,Z 624.122,A -85,B 0,C 180,E1 -5844.782,E2 -5844.782} C_VEL
LIN {X 0,Y 502.228,Z 627.824,A -85,B 0,C 180,E1 -5845.989,E2 -5845.989} C_VEL
LIN {X 0,Y 502.134,Z 629.724,A -85,B 0,C 180,E1 -5846.792,E2 -5846.792} C_VEL
LIN {X 0,Y 502.121,Z 631.152,A -85,B 0,C 180,E1 -5847.594,E2 -5847.594} C_VEL
LIN {X 0,Y 502.014,Z 632.767,A -85,B 0,C 180,E1 -5849.199,E2 -5849.199} C_VEL
LIN {X 0,Y 502.018,Z 632.975,A -85,B 0,C 180,E1 -5850.001,E2 -5850.001} C_VEL
LIN {X 0,Y 502.016,Z 632.741,A -85,B 0,C 180,E1 -5850.803,E2 -5850.803} C_VEL
LIN {X 0,Y 502.039,Z 632.106,A -85,B 0,C 180,E1 -5851.605,E2 -5851.605} C_VEL
LIN {X 0,Y 502.126,Z 631.067,A -85,B 0,C 180,E1 -5852.407,E2 -5852.407} C_VEL
LIN {X 0,Y 502.17,Z 629.608,A -85,B 0,C 180,E1 -5853.21,E2 -5853.21} C_VEL
LIN {X 0,Y 502.158,Z 626.554,A -85,B 0,C 180,E1 -5854.416,E2 -5854.416} C_VEL
LIN {X 0,Y 502.243,Z 622.429,A -85,B 0,C 180,E1 -5855.622,E2 -5855.622} C_VEL
LIN {X 0,Y 502.327,Z 616.186,A -85,B 0,C 180,E1 -5857.012,E2 -5857.012} C_VEL
LIN {X 0,Y 502.44,Z 609.134,A -85,B 0,C 180,E1 -5858.244,E2 -5858.244} C_VEL
LIN {X 0,Y 502.644,Z 600.501,A -85,B 0,C 180,E1 -5859.457,E2 -5859.457} C_VEL
LIN {X 0,Y 502.866,Z 590.598,A -85,B 0,C 180,E1 -5860.571,E2 -5860.571} C_VEL
LIN {X 0,Y 503.199,Z 580.64,A -85,B 0,C 180,E1 -5861.481,E2 -5861.481} C_VEL
LIN {X 0,Y 503.454,Z 570.114,A -85,B 0,C 180,E1 -5862.265,E2 -5862.265} C_VEL
LIN {X 0,Y 503.822,Z 558.505,A -85,B 0,C 180,E1 -5862.949,E2 -5862.949} C_VEL
LIN {X 0,Y 504.13,Z 546.089,A -85,B 0,C 180,E1 -5863.505,E2 -5863.505} C_VEL
LIN {X 0,Y 504.448,Z 532.546,A -85,B 0,C 180,E1 -5863.932,E2 -5863.932} C_VEL
LIN {X 0,Y 504.67,Z 517.451,A -85,B 0,C 180,E1 -5864.209,E2 -5864.209} C_VEL
LIN {X 0,Y 505.151,Z 433.182,A -85,B 0,C 180,E1 -5865.496,E2 -5865.496} C_VEL
LIN {X 0,Y 503.206,Z 417.75,A -85,B 0,C 180,E1 -5865.824,E2 -5865.824} C_VEL
LIN {X 0,Y 503.736,Z 395.784,A -85,B 0,C 180,E1 -5868.929,E2 -5868.929} C_VEL
LIN {X 0,Y 504.36,Z 372.296,A -85,B 0,C 180,E1 -5872.317,E2 -5872.317} C_VEL
LIN {X 0,Y 504.868,Z 355.178,A -85,B 0,C 180,E1 -5874.849,E2 -5874.849} C_VEL
LIN {X 0,Y 503.329,Z 346.071,A -85,B 0,C 180,E1 -5876.317,E2 -5876.317} C_VEL
LIN {X 0,Y 502.859,Z 343.85,A -85,B 0,C 180,E1 -5876.718,E2 -5876.718} C_VEL
LIN {X 0,Y 502.83,Z 343.855,A -85,B 0,C 180,E1 -5879.288,E2 -5879.288} C_VEL
LIN {X 0,Y 502.789,Z 343.854,A -85,B 0,C 180,E1 -5882.085,E2 -5882.085} C_VEL
LIN {X 0,Y 502.807,Z 343.857,A -85,B 0,C 180,E1 -5884.966,E2 -5884.966} C_VEL
LIN {X 0,Y 502.799,Z 343.852,A -85,B 0,C 180,E1 -5887.954,E2 -5887.954} C_VEL
LIN {X 0,Y 502.825,Z 343.854,A -85,B 0,C 180,E1 -5891.066,E2 -5891.066} C_VEL
LIN {X 0,Y 502.806,Z 343.853,A -85,B 0,C 180,E1 -5894.532,E2 -5894.532} C_VEL
LIN {X 0,Y 502.803,Z 343.85,A -85,B 0,C 180,E1 -5897.861,E2 -5897.861} C_VEL
LIN {X 0,Y 502.807,Z 343.856,A -85,B 0,C 180,E1 -5901.024,E2 -5901.024} C_VEL
LIN {X 0,Y 502.78,Z 343.853,A -85,B 0,C 180,E1 -5904.169,E2 -5904.169} C_VEL
LIN {X 0,Y 502.838,Z 343.852,A -85,B 0,C 180,E1 -5906.994,E2 -5906.994} C_VEL
LIN {X 0,Y 502.82,Z 343.849,A -85,B 0,C 180,E1 -5910.065,E2 -5910.065} C_VEL
LIN {X 0,Y 502.838,Z 343.851,A -85,B 0,C 180,E1 -5912.533,E2 -5912.533} C_VEL
LIN {X 0,Y 502.832,Z 343.85,A -85,B 0,C 180,E1 -5915.299,E2 -5915.299} C_VEL
LIN {X 0,Y 502.785,Z 343.855,A -85,B 0,C 180,E1 -5917.827,E2 -5917.827} C_VEL
LIN {X 0,Y 502.829,Z 343.853,A -85,B 0,C 180,E1 -5920.4,E2 -5920.4} C_VEL
LIN {X 0,Y 502.874,Z 344.053,A -85,B 0,C 180,E1 -5922.776,E2 -5922.776} C_VEL
LIN {X 0,Y 503.501,Z 350.247,A -85,B 0,C 180,E1 -5924.316,E2 -5924.316} C_VEL
LIN {X 0,Y 505.404,Z 358.74,A -85,B 0,C 180,E1 -5924.523,E2 -5924.523} C_VEL
LIN {X 0,Y 504.649,Z 455.771,A -85,B 0,C 180,E1 -5926.048,E2 -5926.048} C_VEL
LIN {X 0,Y 504.501,Z 469.366,A -85,B 0,C 180,E1 -5926.429,E2 -5926.429} C_VEL
LIN {X 0,Y 504.218,Z 481.135,A -85,B 0,C 180,E1 -5926.909,E2 -5926.909} C_VEL
LIN {X 0,Y 504.022,Z 492.306,A -85,B 0,C 180,E1 -5927.519,E2 -5927.519} C_VEL
LIN {X 0,Y 503.716,Z 503.849,A -85,B 0,C 180,E1 -5928.328,E2 -5928.328} C_VEL
LIN {X 0,Y 503.387,Z 514.232,A -85,B 0,C 180,E1 -5929.238,E2 -5929.238} C_VEL
LIN {X 0,Y 503.155,Z 522.693,A -85,B 0,C 180,E1 -5930.148,E2 -5930.148} C_VEL
LIN {X 0,Y 502.832,Z 531.816,A -85,B 0,C 180,E1 -5931.358,E2 -5931.358} C_VEL
LIN {X 0,Y 502.601,Z 539.129,A -85,B 0,C 180,E1 -5932.568,E2 -5932.568} C_VEL
LIN {X 0,Y 502.452,Z 544.068,A -85,B 0,C 180,E1 -5933.575,E2 -5933.575} C_VEL
LIN {X 0,Y 502.352,Z 548.838,A -85,B 0,C 180,E1 -5934.782,E2 -5934.782} C_VEL
LIN {X 0,Y 502.311,Z 552.482,A -85,B 0,C 180,E1 -5935.988,E2 -5935.988} C_VEL
LIN {X 0,Y 502.258,Z 554.357,A -85,B 0,C 180,E1 -5936.791,E2 -5936.791} C_VEL
LIN {X 0,Y 502.134,Z 555.788,A -85,B 0,C 180,E1 -5937.593,E2 -5937.593} C_VEL
LIN {X 0,Y 502.047,Z 557.393,A -85,B 0,C 180,E1 -5939.198,E2 -5939.198} C_VEL
LIN {X 0,Y 502.043,Z 557.614,A -85,B 0,C 180,E1 -5940,E2 -5940} C_VEL
LIN {X 0,Y 502.046,Z 557.409,A -85,B 0,C 180,E1 -5940.802,E2 -5940.802} C_VEL
LIN {X 0,Y 502.13,Z 555.795,A -85,B 0,C 180,E1 -5942.406,E2 -5942.406} C_VEL
LIN {X 0,Y 502.25,Z 554.394,A -85,B 0,C 180,E1 -5943.209,E2 -5943.209} C_VEL
LIN {X 0,Y 502.276,Z 551.465,A -85,B 0,C 180,E1 -5944.414,E2 -5944.414} C_VEL
LIN {X 0,Y 502.303,Z 547.499,A -85,B 0,C 180,E1 -5945.621,E2 -5945.621} C_VEL
LIN {X 0,Y 502.502,Z 541.556,A -85,B 0,C 180,E1 -5946.992,E2 -5946.992} C_VEL
LIN {X 0,Y 502.698,Z 534.667,A -85,B 0,C 180,E1 -5948.239,E2 -5948.239} C_VEL
LIN {X 0,Y 502.946,Z 526.333,A -85,B 0,C 180,E1 -5949.45,E2 -5949.45} C_VEL
LIN {X 0,Y 503.233,Z 517.73,A -85,B 0,C 180,E1 -5950.46,E2 -5950.46} C_VEL
LIN {X 0,Y 503.59,Z 507.108,A -85,B 0,C 180,E1 -5951.471,E2 -5951.471} C_VEL
LIN {X 0,Y 503.908,Z 495.982,A -85,B 0,C 180,E1 -5952.32,E2 -5952.32} C_VEL
LIN {X 0,Y 504.153,Z 484.818,A -85,B 0,C 180,E1 -5952.99,E2 -5952.99} C_VEL
LIN {X 0,Y 504.461,Z 472.631,A -85,B 0,C 180,E1 -5953.546,E2 -5953.546} C_VEL
LIN {X 0,Y 504.669,Z 460.26,A -85,B 0,C 180,E1 -5953.951,E2 -5953.951} C_VEL
LIN {X 0,Y 504.782,Z 446.307,A -85,B 0,C 180,E1 -5954.231,E2 -5954.231} C_VEL
LIN {X 0,Y 505.386,Z 358.733,A -85,B 0,C 180,E1 -5955.56,E2 -5955.56} C_VEL
LIN {X 0,Y 503.239,Z 348.163,A -85,B 0,C 180,E1 -5955.814,E2 -5955.814} C_VEL
LIN {X 0,Y 502.865,Z 343.849,A -85,B 0,C 180,E1 -5956.858,E2 -5956.858} C_VEL
LIN {X 0,Y 502.828,Z 343.853,A -85,B 0,C 180,E1 -5959.6,E2 -5959.6} C_VEL
LIN {X 0,Y 502.808,Z 343.852,A -85,B 0,C 180,E1 -5962.702,E2 -5962.702} C_VEL
LIN {X 0,Y 502.843,Z 343.849,A -85,B 0,C 180,E1 -5965.675,E2 -5965.675} C_VEL
LIN {X 0,Y 502.845,Z 343.846,A -85,B 0,C 180,E1 -5968.372,E2 -5968.372} C_VEL
LIN {X 0,Y 502.797,Z 343.856,A -85,B 0,C 180,E1 -5971.498,E2 -5971.498} C_VEL
LIN {X 0,Y 502.808,Z 343.85,A -85,B 0,C 180,E1 -5973.994,E2 -5973.994} C_VEL
LIN {X 0,Y 502.782,Z 343.858,A -85,B 0,C 180,E1 -5977.177,E2 -5977.177} C_VEL
LIN {X 0,Y 502.792,Z 343.852,A -85,B 0,C 180,E1 -5980.015,E2 -5980.015} C_VEL
LIN {X 0,Y 502.8,Z 343.851,A -85,B 0,C 180,E1 -5982.11,E2 -5982.11} C_VEL
LIN {X 0,Y 502.162,Z 343.935,A -85,B 0,C 180,E1 -5982.779,E2 -5982.779} C_VEL
LIN {X 0,Y 499.3,Z 344.292,A -85,B 0,C 180,E1 -5983.863,E2 -5983.863} C_VEL
LIN {X 0,Y 496.862,Z 344.595,A -85,B 0,C 180,E1 -5984.737,E2 -5984.737} C_VEL
LIN {X 0,Y 495.815,Z 344.725,A -85,B 0,C 180,E1 -5985.412,E2 -5985.412} C_VEL
LIN {X 0,Y 495.731,Z 344.732,A -85,B 0,C 180,E1 -5985.641,E2 -5985.641} C_VEL
LIN {X 0,Y 495.759,Z 344.733,A -85,B 0,C 180,E1 -5988.707,E2 -5988.707} C_VEL
LIN {X 0,Y 495.756,Z 344.732,A -85,B 0,C 180,E1 -5991.408,E2 -5991.408} C_VEL
LIN {X 0,Y 495.754,Z 344.731,A -85,B 0,C 180,E1 -5994.462,E2 -5994.462} C_VEL
LIN {X 0,Y 495.772,Z 344.729,A -85,B 0,C 180,E1 -5997.405,E2 -5997.405} C_VEL
LIN {X 0,Y 495.771,Z 344.728,A -85,B 0,C 180,E1 -6000.253,E2 -6000.253} C_VEL
LIN {X 0,Y 495.828,Z 344.723,A -85,B 0,C 180,E1 -6003.25,E2 -6003.25} C_VEL
LIN {X 0,Y 495.757,Z 344.729,A -85,B 0,C 180,E1 -6005.724,E2 -6005.724} C_VEL
LIN {X 0,Y 495.747,Z 344.733,A -85,B 0,C 180,E1 -6008.37,E2 -6008.37} C_VEL
LIN {X 0,Y 495.788,Z 344.728,A -85,B 0,C 180,E1 -6010.971,E2 -6010.971} C_VEL
LIN {X 0,Y 495.783,Z 344.725,A -85,B 0,C 180,E1 -6013.529,E2 -6013.529} C_VEL
LIN {X 0,Y 495.798,Z 344.724,A -85,B 0,C 180,E1 -6016.055,E2 -6016.055} C_VEL
LIN {X 0,Y 495.855,Z 344.722,A -85,B 0,C 180,E1 -6018.554,E2 -6018.554} C_VEL
LIN {X 0,Y 495.876,Z 344.714,A -85,B 0,C 180,E1 -6021.851,E2 -6021.851} C_VEL
LIN {X 0,Y 495.893,Z 344.716,A -85,B 0,C 180,E1 -6024.306,E2 -6024.306} C_VEL
LIN {X 0,Y 495.997,Z 344.698,A -85,B 0,C 180,E1 -6027.563,E2 -6027.563} C_VEL
LIN {X 0,Y 496.001,Z 344.7,A -85,B 0,C 180,E1 -6029.999,E2 -6029.999} C_VEL
LIN {X 0,Y 495.997,Z 344.704,A -85,B 0,C 180,E1 -6032.435,E2 -6032.435} C_VEL
LIN {X 0,Y 495.901,Z 344.711,A -85,B 0,C 180,E1 -6035.692,E2 -6035.692} C_VEL
LIN {X 0,Y 495.874,Z 344.718,A -85,B 0,C 180,E1 -6038.147,E2 -6038.147} C_VEL
LIN {X 0,Y 495.852,Z 344.716,A -85,B 0,C 180,E1 -6041.444,E2 -6041.444} C_VEL
LIN {X 0,Y 495.79,Z 344.727,A -85,B 0,C 180,E1 -6044.782,E2 -6044.782} C_VEL
LIN {X 0,Y 495.788,Z 344.724,A -85,B 0,C 180,E1 -6047.317,E2 -6047.317} C_VEL
LIN {X 0,Y 495.777,Z 344.728,A -85,B 0,C 180,E1 -6049.889,E2 -6049.889} C_VEL
LIN {X 0,Y 495.756,Z 344.73,A -85,B 0,C 180,E1 -6052.859,E2 -6052.859} C_VEL
LIN {X 0,Y 495.798,Z 344.729,A -85,B 0,C 180,E1 -6056.066,E2 -6056.066} C_VEL
LIN {X 0,Y 495.778,Z 344.727,A -85,B 0,C 180,E1 -6058.813,E2 -6058.813} C_VEL
LIN {X 0,Y 495.756,Z 344.731,A -85,B 0,C 180,E1 -6061.725,E2 -6061.725} C_VEL
LIN {X 0,Y 495.773,Z 344.727,A -85,B 0,C 180,E1 -6064.694,E2 -6064.694} C_VEL
LIN {X 0,Y 495.728,Z 344.733,A -85,B 0,C 180,E1 -6067.56,E2 -6067.56} C_VEL
LIN {X 0,Y 495.795,Z 344.73,A -85,B 0,C 180,E1 -6070.052,E2 -6070.052} C_VEL
LIN {X 0,Y 495.756,Z 344.728,A -85,B 0,C 180,E1 -6072.878,E2 -6072.878} C_VEL
LIN {X 0,Y 495.731,Z 344.738,A -85,B 0,C 180,E1 -6075.999,E2 -6075.999} C_VEL
LIN {X 0,Y 495.767,Z 344.727,A -85,B 0,C 180,E1 -6078.704,E2 -6078.704} C_VEL
LIN {X 0,Y 495.756,Z 344.729,A -85,B 0,C 180,E1 -6081.409,E2 -6081.409} C_VEL
LIN {X 0,Y 495.75,Z 344.73,A -85,B 0,C 180,E1 -6084.462,E2 -6084.462} C_VEL
LIN {X 0,Y 495.761,Z 344.729,A -85,B 0,C 180,E1 -6087.405,E2 -6087.405} C_VEL
LIN {X 0,Y 495.773,Z 344.728,A -85,B 0,C 180,E1 -6090.254,E2 -6090.254} C_VEL
LIN {X 0,Y 495.825,Z 344.72,A -85,B 0,C 180,E1 -6093.248,E2 -6093.248} C_VEL
LIN {X 0,Y 495.744,Z 344.736,A -85,B 0,C 180,E1 -6095.725,E2 -6095.725} C_VEL
LIN {X 0,Y 495.735,Z 344.731,A -85,B 0,C 180,E1 -6098.371,E2 -6098.371} C_VEL
LIN {X 0,Y 495.776,Z 344.725,A -85,B 0,C 180,E1 -6100.971,E2 -6100.971} C_VEL
LIN {X 0,Y 495.772,Z 344.731,A -85,B 0,C 180,E1 -6103.53,E2 -6103.53} C_VEL
LIN {X 0,Y 495.785,Z 344.727,A -85,B 0,C 180,E1 -6106.055,E2 -6106.055} C_VEL
LIN {X 0,Y 495.86,Z 344.714,A -85,B 0,C 180,E1 -6108.555,E2 -6108.555} C_VEL
LIN {X 0,Y 495.864,Z 344.718,A -85,B 0,C 180,E1 -6111.852,E2 -6111.852} C_VEL
LIN {X 0,Y 495.887,Z 344.711,A -85,B 0,C 180,E1 -6114.307,E2 -6114.307} C_VEL
LIN {X 0,Y 495.985,Z 344.707,A -85,B 0,C 180,E1 -6117.564,E2 -6117.564} C_VEL
LIN {X 0,Y 495.988,Z 344.7,A -85,B 0,C 180,E1 -6120,E2 -6120} C_VEL
LIN {X 0,Y 495.985,Z 344.698,A -85,B 0,C 180,E1 -6122.436,E2 -6122.436} C_VEL
LIN {X 0,Y 495.904,Z 344.713,A -85,B 0,C 180,E1 -6125.693,E2 -6125.693} C_VEL
LIN {X 0,Y 495.864,Z 344.714,A -85,B 0,C 180,E1 -6128.148,E2 -6128.148} C_VEL
LIN {X 0,Y 495.86,Z 344.722,A -85,B 0,C 180,E1 -6131.445,E2 -6131.445} C_VEL
LIN {X 0,Y 495.781,Z 344.725,A -85,B 0,C 180,E1 -6134.783,E2 -6134.783} C_VEL
LIN {X 0,Y 495.78,Z 344.732,A -85,B 0,C 180,E1 -6137.319,E2 -6137.319} C_VEL
LIN {X 0,Y 495.77,Z 344.727,A -85,B 0,C 180,E1 -6139.891,E2 -6139.891} C_VEL
LIN {X 0,Y 495.757,Z 344.73,A -85,B 0,C 180,E1 -6142.863,E2 -6142.863} C_VEL
LIN {X 0,Y 495.791,Z 344.723,A -85,B 0,C 180,E1 -6146.068,E2 -6146.068} C_VEL
LIN {X 0,Y 495.764,Z 344.729,A -85,B 0,C 180,E1 -6148.815,E2 -6148.815} C_VEL
LIN {X 0,Y 495.751,Z 344.729,A -85,B 0,C 180,E1 -6151.727,E2 -6151.727} C_VEL
LIN {X 0,Y 495.77,Z 344.728,A -85,B 0,C 180,E1 -6154.696,E2 -6154.696} C_VEL
LIN {X 0,Y 495.728,Z 344.733,A -85,B 0,C 180,E1 -6157.562,E2 -6157.562} C_VEL
LIN {X 0,Y 495.788,Z 344.723,A -85,B 0,C 180,E1 -6160.053,E2 -6160.053} C_VEL
LIN {X 0,Y 495.759,Z 344.732,A -85,B 0,C 180,E1 -6162.88,E2 -6162.88} C_VEL
LIN {X 0,Y 495.731,Z 344.73,A -85,B 0,C 180,E1 -6166,E2 -6166} C_VEL
LIN {X 0,Y 495.763,Z 344.73,A -85,B 0,C 180,E1 -6168.706,E2 -6168.706} C_VEL
LIN {X 0,Y 495.761,Z 344.73,A -85,B 0,C 180,E1 -6171.411,E2 -6171.411} C_VEL
LIN {X 0,Y 495.755,Z 344.73,A -85,B 0,C 180,E1 -6174.464,E2 -6174.464} C_VEL
LIN {X 0,Y 495.767,Z 344.728,A -85,B 0,C 180,E1 -6177.407,E2 -6177.407} C_VEL
LIN {X 0,Y 495.78,Z 344.729,A -85,B 0,C 180,E1 -6180.256,E2 -6180.256} C_VEL
LIN {X 0,Y 495.822,Z 344.763,A -85,B 0,C 180,E1 -6182.828,E2 -6182.828} C_VEL
LIN {X 0,Y 498.177,Z 356.283,A -85,B 0,C 180,E1 -6184.716,E2 -6184.716} C_VEL
LIN {X 0,Y 498.115,Z 363.731,A -85,B 0,C 180,E1 -6185.849,E2 -6185.849} C_VEL
LIN {X 0,Y 497.375,Z 383.862,A -85,B 0,C 180,E1 -6188.843,E2 -6188.843} C_VEL
LIN {X 0,Y 496.708,Z 405.927,A -85,B 0,C 180,E1 -6192.078,E2 -6192.078} C_VEL
LIN {X 0,Y 496.337,Z 418.955,A -85,B 0,C 180,E1 -6193.97,E2 -6193.97} C_VEL
LIN {X 0,Y 498.385,Z 434.242,A -85,B 0,C 180,E1 -6194.287,E2 -6194.287} C_VEL
LIN {X 0,Y 497.721,Z 528.118,A -85,B 0,C 180,E1 -6195.747,E2 -6195.747} C_VEL
LIN {X 0,Y 497.386,Z 541.935,A -85,B 0,C 180,E1 -6196.128,E2 -6196.128} C_VEL
LIN {X 0,Y 497.021,Z 554.959,A -85,B 0,C 180,E1 -6196.665,E2 -6196.665} C_VEL
LIN {X 0,Y 496.675,Z 567.465,A -85,B 0,C 180,E1 -6197.373,E2 -6197.373} C_VEL
LIN {X 0,Y 496.33,Z 578.283,A -85,B 0,C 180,E1 -6198.153,E2 -6198.153} C_VEL
LIN {X 0,Y 496.017,Z 588.631,A -85,B 0,C 180,E1 -6199.077,E2 -6199.077} C_VEL
LIN {X 0,Y 495.632,Z 598.749,A -85,B 0,C 180,E1 -6200.204,E2 -6200.204} C_VEL
LIN {X 0,Y 495.422,Z 607.673,A -85,B 0,C 180,E1 -6201.435,E2 -6201.435} C_VEL
LIN {X 0,Y 495.264,Z 614.787,A -85,B 0,C 180,E1 -6202.664,E2 -6202.664} C_VEL
LIN {X 0,Y 495.115,Z 621.035,A -85,B 0,C 180,E1 -6204.03,E2 -6204.03} C_VEL
LIN {X 0,Y 495.039,Z 624.925,A -85,B 0,C 180,E1 -6205.115,E2 -6205.115} C_VEL
LIN {X 0,Y 495.134,Z 627.285,A -85,B 0,C 180,E1 -6205.931,E2 -6205.931} C_VEL
LIN {X 0,Y 495.059,Z 629.192,A -85,B 0,C 180,E1 -6206.746,E2 -6206.746} C_VEL
LIN {X 0,Y 495.055,Z 630.626,A -85,B 0,C 180,E1 -6207.56,E2 -6207.56} C_VEL
LIN {X 0,Y 494.933,Z 632.24,A -85,B 0,C 180,E1 -6209.187,E2 -6209.187} C_VEL
LIN {X 0,Y 494.938,Z 632.447,A -85,B 0,C 180,E1 -6210.001,E2 -6210.001} C_VEL
LIN {X 0,Y 494.935,Z 632.208,A -85,B 0,C 180,E1 -6210.815,E2 -6210.815} C_VEL
LIN {X 0,Y 494.965,Z 631.563,A -85,B 0,C 180,E1 -6211.628,E2 -6211.628} C_VEL
LIN {X 0,Y 495.06,Z 630.516,A -85,B 0,C 180,E1 -6212.442,E2 -6212.442} C_VEL
LIN {X 0,Y 495.092,Z 629.045,A -85,B 0,C 180,E1 -6213.256,E2 -6213.256} C_VEL
LIN {X 0,Y 495.057,Z 625.967,A -85,B 0,C 180,E1 -6214.479,E2 -6214.479} C_VEL
LIN {X 0,Y 495.156,Z 621.815,A -85,B 0,C 180,E1 -6215.703,E2 -6215.703} C_VEL
LIN {X 0,Y 495.247,Z 615.524,A -85,B 0,C 180,E1 -6217.113,E2 -6217.113} C_VEL
LIN {X 0,Y 495.366,Z 608.432,A -85,B 0,C 180,E1 -6218.363,E2 -6218.363} C_VEL
LIN {X 0,Y 495.584,Z 599.742,A -85,B 0,C 180,E1 -6219.593,E2 -6219.593} C_VEL
LIN {X 0,Y 495.869,Z 589.777,A -85,B 0,C 180,E1 -6220.722,E2 -6220.722} C_VEL
LIN {X 0,Y 496.196,Z 579.753,A -85,B 0,C 180,E1 -6221.645,E2 -6221.645} C_VEL
LIN {X 0,Y 496.49,Z 569.051,A -85,B 0,C 180,E1 -6222.446,E2 -6222.446} C_VEL
LIN {X 0,Y 496.876,Z 557.397,A -85,B 0,C 180,E1 -6223.133,E2 -6223.133} C_VEL
LIN {X 0,Y 497.194,Z 544.838,A -85,B 0,C 180,E1 -6223.697,E2 -6223.697} C_VEL
LIN {X 0,Y 497.531,Z 532,A -85,B 0,C 180,E1 -6224.104,E2 -6224.104} C_VEL
LIN {X 0,Y 497.754,Z 517.031,A -85,B 0,C 180,E1 -6224.385,E2 -6224.385} C_VEL
LIN {X 0,Y 498.314,Z 434.114,A -85,B 0,C 180,E1 -6225.687,E2 -6225.687} C_VEL
LIN {X 0,Y 496.201,Z 417.151,A -85,B 0,C 180,E1 -6226.047,E2 -6226.047} C_VEL
LIN {X 0,Y 496.791,Z 393.774,A -85,B 0,C 180,E1 -6229.418,E2 -6229.418} C_VEL
LIN {X 0,Y 497.406,Z 373.309,A -85,B 0,C 180,E1 -6232.427,E2 -6232.427} C_VEL
LIN {X 0,Y 497.936,Z 355.928,A -85,B 0,C 180,E1 -6235.052,E2 -6235.052} C_VEL
LIN {X 0,Y 495.824,Z 344.727,A -85,B 0,C 180,E1 -6236.936,E2 -6236.936} C_VEL
LIN {X 0,Y 495.771,Z 344.729,A -85,B 0,C 180,E1 -6240.148,E2 -6240.148} C_VEL
LIN {X 0,Y 495.799,Z 344.731,A -85,B 0,C 180,E1 -6243.245,E2 -6243.245} C_VEL
LIN {X 0,Y 495.726,Z 344.733,A -85,B 0,C 180,E1 -6246.089,E2 -6246.089} C_VEL
LIN {X 0,Y 495.77,Z 344.731,A -85,B 0,C 180,E1 -6248.769,E2 -6248.769} C_VEL
LIN {X 0,Y 495.761,Z 344.728,A -85,B 0,C 180,E1 -6251.781,E2 -6251.781} C_VEL
LIN {X 0,Y 495.755,Z 344.734,A -85,B 0,C 180,E1 -6255.14,E2 -6255.14} C_VEL
LIN {X 0,Y 495.763,Z 344.727,A -85,B 0,C 180,E1 -6258.219,E2 -6258.219} C_VEL
LIN {X 0,Y 495.755,Z 344.731,A -85,B 0,C 180,E1 -6261.409,E2 -6261.409} C_VEL
LIN {X 0,Y 495.753,Z 344.73,A -85,B 0,C 180,E1 -6264.462,E2 -6264.462} C_VEL
LIN {X 0,Y 495.773,Z 344.729,A -85,B 0,C 180,E1 -6267.406,E2 -6267.406} C_VEL
LIN {X 0,Y 495.772,Z 344.728,A -85,B 0,C 180,E1 -6270.254,E2 -6270.254} C_VEL
LIN {X 0,Y 495.829,Z 344.724,A -85,B 0,C 180,E1 -6273.251,E2 -6273.251} C_VEL
LIN {X 0,Y 495.753,Z 344.73,A -85,B 0,C 180,E1 -6275.725,E2 -6275.725} C_VEL
LIN {X 0,Y 495.748,Z 344.735,A -85,B 0,C 180,E1 -6278.371,E2 -6278.371} C_VEL
LIN {X 0,Y 495.787,Z 344.731,A -85,B 0,C 180,E1 -6280.972,E2 -6280.972} C_VEL
LIN {X 0,Y 495.834,Z 344.814,A -85,B 0,C 180,E1 -6282.523,E2 -6282.523} C_VEL
LIN {X 0,Y 496.568,Z 350.945,A -85,B 0,C 180,E1 -6284.079,E2 -6284.079} C_VEL
LIN {X 0,Y 498.613,Z 359.627,A -85,B 0,C 180,E1 -6284.307,E2 -6284.307} C_VEL
LIN {X 0,Y 497.767,Z 456.552,A -85,B 0,C 180,E1 -6285.877,E2 -6285.877} C_VEL
LIN {X 0,Y 497.586,Z 470.033,A -85,B 0,C 180,E1 -6286.263,E2 -6286.263} C_VEL
LIN {X 0,Y 497.295,Z 482.309,A -85,B 0,C 180,E1 -6286.775,E2 -6286.775} C_VEL
LIN {X 0,Y 497.074,Z 494.38,A -85,B 0,C 180,E1 -6287.463,E2 -6287.463} C_VEL
LIN {X 0,Y 496.731,Z 505.436,A -85,B 0,C 180,E1 -6288.265,E2 -6288.265} C_VEL
LIN {X 0,Y 496.392,Z 515.625,A -85,B 0,C 180,E1 -6289.187,E2 -6289.187} C_VEL
LIN {X 0,Y 496.105,Z 524.748,A -85,B 0,C 180,E1 -6290.212,E2 -6290.212} C_VEL
LIN {X 0,Y 495.785,Z 533.606,A -85,B 0,C 180,E1 -6291.44,E2 -6291.44} C_VEL
LIN {X 0,Y 495.549,Z 540.692,A -85,B 0,C 180,E1 -6292.667,E2 -6292.667} C_VEL
LIN {X 0,Y 495.357,Z 546.306,A -85,B 0,C 180,E1 -6293.892,E2 -6293.892} C_VEL
LIN {X 0,Y 495.3,Z 550.697,A -85,B 0,C 180,E1 -6295.116,E2 -6295.116} C_VEL
LIN {X 0,Y 495.248,Z 553.007,A -85,B 0,C 180,E1 -6295.931,E2 -6295.931} C_VEL
LIN {X 0,Y 495.206,Z 554.886,A -85,B 0,C 180,E1 -6296.746,E2 -6296.746} C_VEL
LIN {X 0,Y 495.071,Z 556.325,A -85,B 0,C 180,E1 -6297.559,E2 -6297.559} C_VEL
LIN {X 0,Y 494.969,Z 557.93,A -85,B 0,C 180,E1 -6299.186,E2 -6299.186} C_VEL
LIN {X 0,Y 494.964,Z 558.148,A -85,B 0,C 180,E1 -6300,E2 -6300} C_VEL
LIN {X 0,Y 494.966,Z 557.938,A -85,B 0,C 180,E1 -6300.813,E2 -6300.813} C_VEL
LIN {X 0,Y 495.068,Z 556.307,A -85,B 0,C 180,E1 -6302.441,E2 -6302.441} C_VEL
LIN {X 0,Y 495.195,Z 554.894,A -85,B 0,C 180,E1 -6303.254,E2 -6303.254} C_VEL
LIN {X 0,Y 495.224,Z 551.946,A -85,B 0,C 180,E1 -6304.477,E2 -6304.477} C_VEL
LIN {X 0,Y 495.253,Z 547.956,A -85,B 0,C 180,E1 -6305.701,E2 -6305.701} C_VEL
LIN {X 0,Y 495.449,Z 542.142,A -85,B 0,C 180,E1 -6307.059,E2 -6307.059} C_VEL
LIN {X 0,Y 495.677,Z 535.051,A -85,B 0,C 180,E1 -6308.356,E2 -6308.356} C_VEL
LIN {X 0,Y 495.96,Z 526.67,A -85,B 0,C 180,E1 -6309.585,E2 -6309.585} C_VEL
LIN {X 0,Y 496.246,Z 518.016,A -85,B 0,C 180,E1 -6310.609,E2 -6310.609} C_VEL
LIN {X 0,Y 496.649,Z 507.336,A -85,B 0,C 180,E1 -6311.633,E2 -6311.633} C_VEL
LIN {X 0,Y 496.959,Z 496.793,A -85,B 0,C 180,E1 -6312.449,E2 -6312.449} C_VEL
LIN {X 0,Y 497.191,Z 486.789,A -85,B 0,C 180,E1 -6313.071,E2 -6313.071} C_VEL
LIN {X 0,Y 497.51,Z 475.14,A -85,B 0,C 180,E1 -6313.635,E2 -6313.635} C_VEL
LIN {X 0,Y 497.737,Z 461.791,A -85,B 0,C 180,E1 -6314.097,E2 -6314.097} C_VEL
LIN {X 0,Y 497.898,Z 448.843,A -85,B 0,C 180,E1 -6314.379,E2 -6314.379} C_VEL
LIN {X 0,Y 498.445,Z 358.983,A -85,B 0,C 180,E1 -6315.778,E2 -6315.778} C_VEL
LIN {X 0,Y 496.22,Z 348.558,A -85,B 0,C 180,E1 -6316.038,E2 -6316.038} C_VEL
LIN {X 0,Y 495.814,Z 344.728,A -85,B 0,C 180,E1 -6316.946,E2 -6316.946} C_VEL
LIN {X 0,Y 495.775,Z 344.728,A -85,B 0,C 180,E1 -6319.89,E2 -6319.89} C_VEL
LIN {X 0,Y 495.764,Z 344.731,A -85,B 0,C 180,E1 -6322.86,E2 -6322.86} C_VEL
LIN {X 0,Y 495.794,Z 344.724,A -85,B 0,C 180,E1 -6326.068,E2 -6326.068} C_VEL
LIN {X 0,Y 495.777,Z 344.729,A -85,B 0,C 180,E1 -6328.814,E2 -6328.814} C_VEL
LIN {X 0,Y 495.76,Z 344.73,A -85,B 0,C 180,E1 -6331.725,E2 -6331.725} C_VEL
LIN {X 0,Y 495.773,Z 344.729,A -85,B 0,C 180,E1 -6334.694,E2 -6334.694} C_VEL
LIN {X 0,Y 495.733,Z 344.734,A -85,B 0,C 180,E1 -6337.561,E2 -6337.561} C_VEL
LIN {X 0,Y 495.771,Z 344.73,A -85,B 0,C 180,E1 -6340.699,E2 -6340.699} C_VEL
LIN {X 0,Y 495.739,Z 344.731,A -85,B 0,C 180,E1 -6344,E2 -6344} C_VEL
LIN {X 0,Y 495.731,Z 344.732,A -85,B 0,C 180,E1 -6345.641,E2 -6345.641} C_VEL
LIN {X 0,Y 495.065,Z 344.816,A -85,B 0,C 180,E1 -6346.319,E2 -6346.319} C_VEL
LIN {X 0,Y 492.205,Z 345.174,A -85,B 0,C 180,E1 -6347.419,E2 -6347.419} C_VEL
LIN {X 0,Y 489.795,Z 345.473,A -85,B 0,C 180,E1 -6348.306,E2 -6348.306} C_VEL
LIN {X 0,Y 488.773,Z 345.603,A -85,B 0,C 180,E1 -6348.991,E2 -6348.991} C_VEL
LIN {X 0,Y 488.697,Z 345.607,A -85,B 0,C 180,E1 -6349.223,E2 -6349.223} C_VEL
LIN {X 0,Y 488.682,Z 345.611,A -85,B 0,C 180,E1 -6352.278,E2 -6352.278} C_VEL
LIN {X 0,Y 488.729,Z 345.608,A -85,B 0,C 180,E1 -6355.052,E2 -6355.052} C_VEL
LIN {X 0,Y 488.708,Z 345.607,A -85,B 0,C 180,E1 -6358.045,E2 -6358.045} C_VEL
LIN {X 0,Y 488.728,Z 345.61,A -85,B 0,C 180,E1 -6360.729,E2 -6360.729} C_VEL
LIN {X 0,Y 488.761,Z 345.601,A -85,B 0,C 180,E1 -6363.527,E2 -6363.527} C_VEL
LIN {X 0,Y 488.697,Z 345.61,A -85,B 0,C 180,E1 -6366.254,E2 -6366.254} C_VEL
LIN {X 0,Y 488.75,Z 345.605,A -85,B 0,C 180,E1 -6369.175,E2 -6369.175} C_VEL
LIN {X 0,Y 488.738,Z 345.607,A -85,B 0,C 180,E1 -6372.423,E2 -6372.423} C_VEL
LIN {X 0,Y 488.766,Z 345.603,A -85,B 0,C 180,E1 -6374.999,E2 -6374.999} C_VEL
LIN {X 0,Y 488.809,Z 345.599,A -85,B 0,C 180,E1 -6378.387,E2 -6378.387} C_VEL
LIN {X 0,Y 488.821,Z 345.593,A -85,B 0,C 180,E1 -6381.733,E2 -6381.733} C_VEL
LIN {X 0,Y 488.851,Z 345.592,A -85,B 0,C 180,E1 -6384.223,E2 -6384.223} C_VEL
LIN {X 0,Y 488.964,Z 345.574,A -85,B 0,C 180,E1 -6387.528,E2 -6387.528} C_VEL
LIN {X 0,Y 488.957,Z 345.579,A -85,B 0,C 180,E1 -6390.823,E2 -6390.823} C_VEL
LIN {X 0,Y 488.964,Z 345.58,A -85,B 0,C 180,E1 -6392.47,E2 -6392.47} C_VEL
LIN {X 0,Y 488.86,Z 345.588,A -85,B 0,C 180,E1 -6395.775,E2 -6395.775} C_VEL
LIN {X 0,Y 488.819,Z 345.599,A -85,B 0,C 180,E1 -6398.265,E2 -6398.265} C_VEL
LIN {X 0,Y 488.806,Z 345.594,A -85,B 0,C 180,E1 -6401.611,E2 -6401.611} C_VEL
LIN {X 0,Y 488.762,Z 345.601,A -85,B 0,C 180,E1 -6404.999,E2 -6404.999} C_VEL
LIN {X 0,Y 488.754,Z 345.605,A -85,B 0,C 180,E1 -6408.441,E2 -6408.441} C_VEL
LIN {X 0,Y 488.706,Z 345.607,A -85,B 0,C 180,E1 -6411.07,E2 -6411.07} C_VEL
LIN {X 0,Y 488.692,Z 345.61,A -85,B 0,C 180,E1 -6413.744,E2 -6413.744} C_VEL
LIN {X 0,Y 488.796,Z 345.596,A -85,B 0,C 180,E1 -6416.944,E2 -6416.944} C_VEL
LIN {X 0,Y 488.716,Z 345.609,A -85,B 0,C 180,E1 -6420.364,E2 -6420.364} C_VEL
LIN {X 0,Y 488.732,Z 345.604,A -85,B 0,C 180,E1 -6423.484,E2 -6423.484} C_VEL
LIN {X 0,Y 488.685,Z 345.613,A -85,B 0,C 180,E1 -6426.355,E2 -6426.355} C_VEL
LIN {X 0,Y 488.745,Z 345.601,A -85,B 0,C 180,E1 -6429.248,E2 -6429.248} C_VEL
LIN {X 0,Y 488.724,Z 345.606,A -85,B 0,C 180,E1 -6431.602,E2 -6431.602} C_VEL
LIN {X 0,Y 488.696,Z 345.614,A -85,B 0,C 180,E1 -6434.023,E2 -6434.023} C_VEL
LIN {X 0,Y 488.739,Z 345.602,A -85,B 0,C 180,E1 -6437.168,E2 -6437.168} C_VEL
LIN {X 0,Y 488.762,Z 345.603,A -85,B 0,C 180,E1 -6439.679,E2 -6439.679} C_VEL
LIN {X 0,Y 488.676,Z 345.61,A -85,B 0,C 180,E1 -6442.841,E2 -6442.841} C_VEL
LIN {X 0,Y 488.727,Z 345.61,A -85,B 0,C 180,E1 -6445.887,E2 -6445.887} C_VEL
LIN {X 0,Y 488.688,Z 345.608,A -85,B 0,C 180,E1 -6448.82,E2 -6448.82} C_VEL
LIN {X 0,Y 488.738,Z 345.608,A -85,B 0,C 180,E1 -6451.671,E2 -6451.671} C_VEL
LIN {X 0,Y 488.742,Z 345.602,A -85,B 0,C 180,E1 -6454.444,E2 -6454.444} C_VEL
LIN {X 0,Y 488.718,Z 345.605,A -85,B 0,C 180,E1 -6457.153,E2 -6457.153} C_VEL
LIN {X 0,Y 488.719,Z 345.61,A -85,B 0,C 180,E1 -6459.81,E2 -6459.81} C_VEL
LIN {X 0,Y 488.726,Z 345.604,A -85,B 0,C 180,E1 -6462.423,E2 -6462.423} C_VEL
LIN {X 0,Y 488.752,Z 345.6,A -85,B 0,C 180,E1 -6464.999,E2 -6464.999} C_VEL
LIN {X 0,Y 488.821,Z 345.591,A -85,B 0,C 180,E1 -6468.388,E2 -6468.388} C_VEL
LIN {X 0,Y 488.809,Z 345.599,A -85,B 0,C 180,E1 -6471.734,E2 -6471.734} C_VEL
LIN {X 0,Y 488.847,Z 345.589,A -85,B 0,C 180,E1 -6474.224,E2 -6474.224} C_VEL
LIN {X 0,Y 488.953,Z 345.583,A -85,B 0,C 180,E1 -6477.529,E2 -6477.529} C_VEL
LIN {X 0,Y 488.96,Z 345.576,A -85,B 0,C 180,E1 -6480,E2 -6480} C_VEL
LIN {X 0,Y 488.953,Z 345.574,A -85,B 0,C 180,E1 -6482.471,E2 -6482.471} C_VEL
LIN {X 0,Y 488.86,Z 345.59,A -85,B 0,C 180,E1 -6485.776,E2 -6485.776} C_VEL
LIN {X 0,Y 488.808,Z 345.592,A -85,B 0,C 180,E1 -6488.267,E2 -6488.267} C_VEL
LIN {X 0,Y 488.821,Z 345.596,A -85,B 0,C 180,E1 -6491.612,E2 -6491.612} C_VEL
LIN {X 0,Y 488.753,Z 345.603,A -85,B 0,C 180,E1 -6495.001,E2 -6495.001} C_VEL
LIN {X 0,Y 488.746,Z 345.6,A -85,B 0,C 180,E1 -6498.443,E2 -6498.443} C_VEL
LIN {X 0,Y 488.698,Z 345.611,A -85,B 0,C 180,E1 -6501.071,E2 -6501.071} C_VEL
LIN {X 0,Y 488.685,Z 345.61,A -85,B 0,C 180,E1 -6503.746,E2 -6503.746} C_VEL
LIN {X 0,Y 488.791,Z 345.599,A -85,B 0,C 180,E1 -6506.946,E2 -6506.946} C_VEL
LIN {X 0,Y 488.702,Z 345.606,A -85,B 0,C 180,E1 -6510.364,E2 -6510.364} C_VEL
LIN {X 0,Y 488.729,Z 345.607,A -85,B 0,C 180,E1 -6513.485,E2 -6513.485} C_VEL
LIN {X 0,Y 488.683,Z 345.609,A -85,B 0,C 180,E1 -6516.357,E2 -6516.357} C_VEL
LIN {X 0,Y 488.743,Z 345.607,A -85,B 0,C 180,E1 -6519.251,E2 -6519.251} C_VEL
LIN {X 0,Y 488.728,Z 345.605,A -85,B 0,C 180,E1 -6522.522,E2 -6522.522} C_VEL
LIN {X 0,Y 488.706,Z 345.612,A -85,B 0,C 180,E1 -6525.2,E2 -6525.2} C_VEL
LIN {X 0,Y 488.73,Z 345.605,A -85,B 0,C 180,E1 -6527.48,E2 -6527.48} C_VEL
LIN {X 0,Y 488.745,Z 345.605,A -85,B 0,C 180,E1 -6530.752,E2 -6530.752} C_VEL
LIN {X 0,Y 488.683,Z 345.609,A -85,B 0,C 180,E1 -6533.87,E2 -6533.87} C_VEL
LIN {X 0,Y 488.737,Z 345.608,A -85,B 0,C 180,E1 -6536.879,E2 -6536.879} C_VEL
LIN {X 0,Y 488.733,Z 345.606,A -85,B 0,C 180,E1 -6539.783,E2 -6539.783} C_VEL
LIN {X 0,Y 488.818,Z 345.755,A -85,B 0,C 180,E1 -6542.638,E2 -6542.638} C_VEL
LIN {X 0,Y 491.407,Z 358.943,A -85,B 0,C 180,E1 -6544.82,E2 -6544.82} C_VEL
LIN {X 0,Y 490.664,Z 379.327,A -85,B 0,C 180,E1 -6547.916,E2 -6547.916} C_VEL
LIN {X 0,Y 489.81,Z 401.756,A -85,B 0,C 180,E1 -6551.262,E2 -6551.262} C_VEL
LIN {X 0,Y 489.34,Z 418.521,A -85,B 0,C 180,E1 -6553.736,E2 -6553.736} C_VEL
LIN {X 0,Y 491.546,Z 435.564,A -85,B 0,C 180,E1 -6554.092,E2 -6554.092} C_VEL
LIN {X 0,Y 490.795,Z 527.963,A -85,B 0,C 180,E1 -6555.568,E2 -6555.568} C_VEL
LIN {X 0,Y 490.441,Z 541.641,A -85,B 0,C 180,E1 -6555.954,E2 -6555.954} C_VEL
LIN {X 0,Y 490.067,Z 554.074,A -85,B 0,C 180,E1 -6556.472,E2 -6556.472} C_VEL
LIN {X 0,Y 489.712,Z 566.04,A -85,B 0,C 180,E1 -6557.149,E2 -6557.149} C_VEL
LIN {X 0,Y 489.385,Z 575.946,A -85,B 0,C 180,E1 -6557.853,E2 -6557.853} C_VEL
LIN {X 0,Y 489.092,Z 585.789,A -85,B 0,C 180,E1 -6558.711,E2 -6558.711} C_VEL
LIN {X 0,Y 488.676,Z 596.452,A -85,B 0,C 180,E1 -6559.854,E2 -6559.854} C_VEL
LIN {X 0,Y 488.379,Z 605.679,A -85,B 0,C 180,E1 -6561.102,E2 -6561.102} C_VEL
LIN {X 0,Y 488.184,Z 613.115,A -85,B 0,C 180,E1 -6562.349,E2 -6562.349} C_VEL
LIN {X 0,Y 488.092,Z 618.556,A -85,B 0,C 180,E1 -6563.478,E2 -6563.478} C_VEL
LIN {X 0,Y 488.05,Z 623.022,A -85,B 0,C 180,E1 -6564.63,E2 -6564.63} C_VEL
LIN {X 0,Y 488.024,Z 626.745,A -85,B 0,C 180,E1 -6565.872,E2 -6565.872} C_VEL
LIN {X 0,Y 487.985,Z 628.66,A -85,B 0,C 180,E1 -6566.698,E2 -6566.698} C_VEL
LIN {X 0,Y 487.99,Z 630.101,A -85,B 0,C 180,E1 -6567.525,E2 -6567.525} C_VEL
LIN {X 0,Y 487.855,Z 631.714,A -85,B 0,C 180,E1 -6569.176,E2 -6569.176} C_VEL
LIN {X 0,Y 487.858,Z 631.918,A -85,B 0,C 180,E1 -6570.001,E2 -6570.001} C_VEL
LIN {X 0,Y 487.857,Z 631.675,A -85,B 0,C 180,E1 -6570.826,E2 -6570.826} C_VEL
LIN {X 0,Y 487.997,Z 629.965,A -85,B 0,C 180,E1 -6572.477,E2 -6572.477} C_VEL
LIN {X 0,Y 488.016,Z 628.481,A -85,B 0,C 180,E1 -6573.303,E2 -6573.303} C_VEL
LIN {X 0,Y 487.962,Z 625.38,A -85,B 0,C 180,E1 -6574.544,E2 -6574.544} C_VEL
LIN {X 0,Y 488.069,Z 621.199,A -85,B 0,C 180,E1 -6575.786,E2 -6575.786} C_VEL
LIN {X 0,Y 488.18,Z 614.758,A -85,B 0,C 180,E1 -6577.238,E2 -6577.238} C_VEL
LIN {X 0,Y 488.304,Z 607.731,A -85,B 0,C 180,E1 -6578.484,E2 -6578.484} C_VEL
LIN {X 0,Y 488.513,Z 598.979,A -85,B 0,C 180,E1 -6579.733,E2 -6579.733} C_VEL
LIN {X 0,Y 488.871,Z 588.966,A -85,B 0,C 180,E1 -6580.877,E2 -6580.877} C_VEL
LIN {X 0,Y 489.193,Z 579.113,A -85,B 0,C 180,E1 -6581.794,E2 -6581.794} C_VEL
LIN {X 0,Y 489.55,Z 567.761,A -85,B 0,C 180,E1 -6582.647,E2 -6582.647} C_VEL
LIN {X 0,Y 489.95,Z 555.309,A -85,B 0,C 180,E1 -6583.375,E2 -6583.375} C_VEL
LIN {X 0,Y 490.318,Z 542.298,A -85,B 0,C 180,E1 -6583.945,E2 -6583.945} C_VEL
LIN {X 0,Y 490.609,Z 529.356,A -85,B 0,C 180,E1 -6584.334,E2 -6584.334} C_VEL
LIN {X 0,Y 490.892,Z 508.459,A -85,B 0,C 180,E1 -6584.696,E2 -6584.696} C_VEL
LIN {X 0,Y 491.431,Z 434.507,A -85,B 0,C 180,E1 -6585.899,E2 -6585.899} C_VEL
LIN {X 0,Y 489.172,Z 416.46,A -85,B 0,C 180,E1 -6586.298,E2 -6586.298} C_VEL
LIN {X 0,Y 489.787,Z 394.704,A -85,B 0,C 180,E1 -6589.489,E2 -6589.489} C_VEL
LIN {X 0,Y 490.453,Z 374.358,A -85,B 0,C 180,E1 -6592.54,E2 -6592.54} C_VEL
LIN {X 0,Y 491.098,Z 358.531,A -85,B 0,C 180,E1 -6594.972,E2 -6594.972} C_VEL
LIN {X 0,Y 489.976,Z 351.356,A -85,B 0,C 180,E1 -6596.172,E2 -6596.172} C_VEL
LIN {X 0,Y 488.773,Z 345.605,A -85,B 0,C 180,E1 -6597.195,E2 -6597.195} C_VEL
LIN {X 0,Y 488.715,Z 345.609,A -85,B 0,C 180,E1 -6600.363,E2 -6600.363} C_VEL
LIN {X 0,Y 488.741,Z 345.608,A -85,B 0,C 180,E1 -6603.485,E2 -6603.485} C_VEL
LIN {X 0,Y 488.688,Z 345.611,A -85,B 0,C 180,E1 -6606.355,E2 -6606.355} C_VEL
LIN {X 0,Y 488.707,Z 345.612,A -85,B 0,C 180,E1 -6609.255,E2 -6609.255} C_VEL
LIN {X 0,Y 488.712,Z 345.607,A -85,B 0,C 180,E1 -6611.6,E2 -6611.6} C_VEL
LIN {X 0,Y 488.718,Z 345.611,A -85,B 0,C 180,E1 -6614.802,E2 -6614.802} C_VEL
LIN {X 0,Y 488.697,Z 345.609,A -85,B 0,C 180,E1 -6617.475,E2 -6617.475} C_VEL
LIN {X 0,Y 488.738,Z 345.604,A -85,B 0,C 180,E1 -6619.677,E2 -6619.677} C_VEL
LIN {X 0,Y 488.685,Z 345.614,A -85,B 0,C 180,E1 -6622.841,E2 -6622.841} C_VEL
LIN {X 0,Y 488.736,Z 345.603,A -85,B 0,C 180,E1 -6625.887,E2 -6625.887} C_VEL
LIN {X 0,Y 488.698,Z 345.614,A -85,B 0,C 180,E1 -6628.82,E2 -6628.82} C_VEL
LIN {X 0,Y 488.75,Z 345.602,A -85,B 0,C 180,E1 -6631.671,E2 -6631.671} C_VEL
LIN {X 0,Y 488.753,Z 345.605,A -85,B 0,C 180,E1 -6634.444,E2 -6634.444} C_VEL
LIN {X 0,Y 488.728,Z 345.609,A -85,B 0,C 180,E1 -6637.153,E2 -6637.153} C_VEL
LIN {X 0,Y 488.73,Z 345.607,A -85,B 0,C 180,E1 -6639.811,E2 -6639.811} C_VEL
LIN {X 0,Y 488.778,Z 345.669,A -85,B 0,C 180,E1 -6642.271,E2 -6642.271} C_VEL
LIN {X 0,Y 489.649,Z 351.726,A -85,B 0,C 180,E1 -6643.839,E2 -6643.839} C_VEL
LIN {X 0,Y 491.851,Z 360.968,A -85,B 0,C 180,E1 -6644.085,E2 -6644.085} C_VEL
LIN {X 0,Y 490.869,Z 457.581,A -85,B 0,C 180,E1 -6645.701,E2 -6645.701} C_VEL
LIN {X 0,Y 490.706,Z 470.899,A -85,B 0,C 180,E1 -6646.093,E2 -6646.093} C_VEL
LIN {X 0,Y 490.369,Z 483.565,A -85,B 0,C 180,E1 -6646.638,E2 -6646.638} C_VEL
LIN {X 0,Y 490.087,Z 496.169,A -85,B 0,C 180,E1 -6647.38,E2 -6647.38} C_VEL
LIN {X 0,Y 489.743,Z 507.066,A -85,B 0,C 180,E1 -6648.2,E2 -6648.2} C_VEL
LIN {X 0,Y 489.438,Z 516.017,A -85,B 0,C 180,E1 -6649.032,E2 -6649.032} C_VEL
LIN {X 0,Y 489.131,Z 525.172,A -85,B 0,C 180,E1 -6650.071,E2 -6650.071} C_VEL
LIN {X 0,Y 488.771,Z 534.067,A -85,B 0,C 180,E1 -6651.316,E2 -6651.316} C_VEL
LIN {X 0,Y 488.522,Z 541.183,A -85,B 0,C 180,E1 -6652.561,E2 -6652.561} C_VEL
LIN {X 0,Y 488.316,Z 546.817,A -85,B 0,C 180,E1 -6653.803,E2 -6653.803} C_VEL
LIN {X 0,Y 488.264,Z 551.22,A -85,B 0,C 180,E1 -6655.045,E2 -6655.045} C_VEL
LIN {X 0,Y 488.188,Z 553.537,A -85,B 0,C 180,E1 -6655.872,E2 -6655.872} C_VEL
LIN {X 0,Y 488.154,Z 555.418,A -85,B 0,C 180,E1 -6656.699,E2 -6656.699} C_VEL
LIN {X 0,Y 488.011,Z 556.862,A -85,B 0,C 180,E1 -6657.524,E2 -6657.524} C_VEL
LIN {X 0,Y 487.89,Z 558.467,A -85,B 0,C 180,E1 -6659.175,E2 -6659.175} C_VEL
LIN {X 0,Y 487.885,Z 558.682,A -85,B 0,C 180,E1 -6660,E2 -6660} C_VEL
LIN {X 0,Y 487.887,Z 558.467,A -85,B 0,C 180,E1 -6660.825,E2 -6660.825} C_VEL
LIN {X 0,Y 488.008,Z 556.817,A -85,B 0,C 180,E1 -6662.476,E2 -6662.476} C_VEL
LIN {X 0,Y 488.142,Z 555.394,A -85,B 0,C 180,E1 -6663.301,E2 -6663.301} C_VEL
LIN {X 0,Y 488.171,Z 552.426,A -85,B 0,C 180,E1 -6664.541,E2 -6664.541} C_VEL
LIN {X 0,Y 488.207,Z 548.411,A -85,B 0,C 180,E1 -6665.783,E2 -6665.783} C_VEL
LIN {X 0,Y 488.429,Z 542.308,A -85,B 0,C 180,E1 -6667.212,E2 -6667.212} C_VEL
LIN {X 0,Y 488.673,Z 535.431,A -85,B 0,C 180,E1 -6668.477,E2 -6668.477} C_VEL
LIN {X 0,Y 488.97,Z 527.002,A -85,B 0,C 180,E1 -6669.723,E2 -6669.723} C_VEL
LIN {X 0,Y 489.265,Z 518.292,A -85,B 0,C 180,E1 -6670.762,E2 -6670.762} C_VEL
LIN {X 0,Y 489.71,Z 507.553,A -85,B 0,C 180,E1 -6671.801,E2 -6671.801} C_VEL
LIN {X 0,Y 490.057,Z 496.164,A -85,B 0,C 180,E1 -6672.68,E2 -6672.68} C_VEL
LIN {X 0,Y 490.336,Z 484.878,A -85,B 0,C 180,E1 -6673.363,E2 -6673.363} C_VEL
LIN {X 0,Y 490.687,Z 472.436,A -85,B 0,C 180,E1 -6673.934,E2 -6673.934} C_VEL
LIN {X 0,Y 490.918,Z 459.567,A -85,B 0,C 180,E1 -6674.35,E2 -6674.35} C_VEL
LIN {X 0,Y 491.009,Z 442.854,A -85,B 0,C 180,E1 -6674.665,E2 -6674.665} C_VEL
LIN {X 0,Y 491.722,Z 360.393,A -85,B 0,C 180,E1 -6675.975,E2 -6675.975} C_VEL
LIN {X 0,Y 489.216,Z 348.971,A -85,B 0,C 180,E1 -6676.269,E2 -6676.269} C_VEL
LIN {X 0,Y 488.765,Z 345.606,A -85,B 0,C 180,E1 -6677.09,E2 -6677.09} C_VEL
LIN {X 0,Y 488.73,Z 345.604,A -85,B 0,C 180,E1 -6680.189,E2 -6680.189} C_VEL
LIN {X 0,Y 488.713,Z 345.611,A -85,B 0,C 180,E1 -6683.02,E2 -6683.02} C_VEL
LIN {X 0,Y 488.743,Z 345.607,A -85,B 0,C 180,E1 -6685.556,E2 -6685.556} C_VEL
LIN {X 0,Y 488.749,Z 345.602,A -85,B 0,C 180,E1 -6688.328,E2 -6688.328} C_VEL
LIN {X 0,Y 488.697,Z 345.612,A -85,B 0,C 180,E1 -6691.179,E2 -6691.179} C_VEL
LIN {X 0,Y 488.735,Z 345.604,A -85,B 0,C 180,E1 -6694.112,E2 -6694.112} C_VEL
LIN {X 0,Y 488.684,Z 345.614,A -85,B 0,C 180,E1 -6697.159,E2 -6697.159} C_VEL
LIN {X 0,Y 488.723,Z 345.606,A -85,B 0,C 180,E1 -6700.344,E2 -6700.344} C_VEL
LIN {X 0,Y 488.692,Z 345.61,A -85,B 0,C 180,E1 -6703.654,E2 -6703.654} C_VEL
LIN {X 0,Y 488.691,Z 345.61,A -85,B 0,C 180,E1 -6706.345,E2 -6706.345} C_VEL
LIN {X 0,Y 488.697,Z 345.607,A -85,B 0,C 180,E1 -6709.223,E2 -6709.223} C_VEL
LIN {X 0,Y 488.042,Z 345.691,A -85,B 0,C 180,E1 -6709.911,E2 -6709.911} C_VEL
LIN {X 0,Y 485.167,Z 346.052,A -85,B 0,C 180,E1 -6711.027,E2 -6711.027} C_VEL
LIN {X 0,Y 482.731,Z 346.352,A -85,B 0,C 180,E1 -6711.927,E2 -6711.927} C_VEL
LIN {X 0,Y 481.693,Z 346.485,A -85,B 0,C 180,E1 -6712.622,E2 -6712.622} C_VEL
LIN {X 0,Y 481.613,Z 346.491,A -85,B 0,C 180,E1 -6712.858,E2 -6712.858} C_VEL
LIN {X 0,Y 481.694,Z 346.484,A -85,B 0,C 180,E1 -6715.317,E2 -6715.317} C_VEL
LIN {X 0,Y 481.649,Z 346.488,A -85,B 0,C 180,E1 -6718.311,E2 -6718.311} C_VEL
LIN {X 0,Y 481.704,Z 346.483,A -85,B 0,C 180,E1 -6721.218,E2 -6721.218} C_VEL
LIN {X 0,Y 481.705,Z 346.48,A -85,B 0,C 180,E1 -6724.042,E2 -6724.042} C_VEL
LIN {X 0,Y 481.678,Z 346.487,A -85,B 0,C 180,E1 -6726.811,E2 -6726.811} C_VEL
LIN {X 0,Y 481.699,Z 346.48,A -85,B 0,C 180,E1 -6729.502,E2 -6729.502} C_VEL
LIN {X 0,Y 481.711,Z 346.48,A -85,B 0,C 180,E1 -6732.158,E2 -6732.158} C_VEL
LIN {X 0,Y 481.746,Z 346.478,A -85,B 0,C 180,E1 -6734.775,E2 -6734.775} C_VEL
LIN {X 0,Y 481.754,Z 346.476,A -85,B 0,C 180,E1 -6738.214,E2 -6738.214} C_VEL
LIN {X 0,Y 481.766,Z 346.471,A -85,B 0,C 180,E1 -6741.611,E2 -6741.611} C_VEL
LIN {X 0,Y 481.812,Z 346.468,A -85,B 0,C 180,E1 -6744.139,E2 -6744.139} C_VEL
LIN {X 0,Y 481.931,Z 346.451,A -85,B 0,C 180,E1 -6747.492,E2 -6747.492} C_VEL
LIN {X 0,Y 481.908,Z 346.457,A -85,B 0,C 180,E1 -6750.835,E2 -6750.835} C_VEL
LIN {X 0,Y 481.931,Z 346.455,A -85,B 0,C 180,E1 -6752.506,E2 -6752.506} C_VEL
LIN {X 0,Y 481.821,Z 346.466,A -85,B 0,C 180,E1 -6755.859,E2 -6755.859} C_VEL
LIN {X 0,Y 481.764,Z 346.477,A -85,B 0,C 180,E1 -6758.387,E2 -6758.387} C_VEL
LIN {X 0,Y 481.751,Z 346.474,A -85,B 0,C 180,E1 -6761.784,E2 -6761.784} C_VEL
LIN {X 0,Y 481.742,Z 346.474,A -85,B 0,C 180,E1 -6765.223,E2 -6765.223} C_VEL
LIN {X 0,Y 481.711,Z 346.48,A -85,B 0,C 180,E1 -6768.721,E2 -6768.721} C_VEL
LIN {X 0,Y 481.646,Z 346.486,A -85,B 0,C 180,E1 -6771.393,E2 -6771.393} C_VEL
LIN {X 0,Y 481.676,Z 346.489,A -85,B 0,C 180,E1 -6774.112,E2 -6774.112} C_VEL
LIN {X 0,Y 481.749,Z 346.473,A -85,B 0,C 180,E1 -6777.139,E2 -6777.139} C_VEL
LIN {X 0,Y 481.685,Z 346.483,A -85,B 0,C 180,E1 -6779.739,E2 -6779.739} C_VEL
LIN {X 0,Y 481.67,Z 346.485,A -85,B 0,C 180,E1 -6782.673,E2 -6782.673} C_VEL
LIN {X 0,Y 481.639,Z 346.489,A -85,B 0,C 180,E1 -6785.708,E2 -6785.708} C_VEL
LIN {X 0,Y 481.717,Z 346.477,A -85,B 0,C 180,E1 -6789.354,E2 -6789.354} C_VEL
LIN {X 0,Y 481.668,Z 346.488,A -85,B 0,C 180,E1 -6792.157,E2 -6792.157} C_VEL
LIN {X 0,Y 481.654,Z 346.487,A -85,B 0,C 180,E1 -6794.456,E2 -6794.456} C_VEL
LIN {X 0,Y 481.683,Z 346.481,A -85,B 0,C 180,E1 -6796.845,E2 -6796.845} C_VEL
LIN {X 0,Y 481.706,Z 346.483,A -85,B 0,C 180,E1 -6800.062,E2 -6800.062} C_VEL
LIN {X 0,Y 481.624,Z 346.49,A -85,B 0,C 180,E1 -6803.375,E2 -6803.375} C_VEL
LIN {X 0,Y 481.701,Z 346.481,A -85,B 0,C 180,E1 -6806.329,E2 -6806.329} C_VEL
LIN {X 0,Y 481.65,Z 346.487,A -85,B 0,C 180,E1 -6809.415,E2 -6809.415} C_VEL
LIN {X 0,Y 481.694,Z 346.482,A -85,B 0,C 180,E1 -6812.168,E2 -6812.168} C_VEL
LIN {X 0,Y 481.709,Z 346.477,A -85,B 0,C 180,E1 -6814.969,E2 -6814.969} C_VEL
LIN {X 0,Y 481.644,Z 346.493,A -85,B 0,C 180,E1 -6817.705,E2 -6817.705} C_VEL
LIN {X 0,Y 481.699,Z 346.479,A -85,B 0,C 180,E1 -6820.393,E2 -6820.393} C_VEL
LIN {X 0,Y 481.683,Z 346.481,A -85,B 0,C 180,E1 -6823.034,E2 -6823.034} C_VEL
LIN {X 0,Y 481.681,Z 346.488,A -85,B 0,C 180,E1 -6825.639,E2 -6825.639} C_VEL
LIN {X 0,Y 481.786,Z 346.469,A -85,B 0,C 180,E1 -6828.216,E2 -6828.216} C_VEL
LIN {X 0,Y 481.755,Z 346.479,A -85,B 0,C 180,E1 -6831.612,E2 -6831.612} C_VEL
LIN {X 0,Y 481.807,Z 346.466,A -85,B 0,C 180,E1 -6834.14,E2 -6834.14} C_VEL
LIN {X 0,Y 481.92,Z 346.458,A -85,B 0,C 180,E1 -6837.493,E2 -6837.493} C_VEL
LIN {X 0,Y 481.931,Z 346.451,A -85,B 0,C 180,E1 -6840,E2 -6840} C_VEL
LIN {X 0,Y 481.92,Z 346.45,A -85,B 0,C 180,E1 -6842.508,E2 -6842.508} C_VEL
LIN {X 0,Y 481.819,Z 346.466,A -85,B 0,C 180,E1 -6845.86,E2 -6845.86} C_VEL
LIN {X 0,Y 481.754,Z 346.471,A -85,B 0,C 180,E1 -6848.389,E2 -6848.389} C_VEL
LIN {X 0,Y 481.786,Z 346.47,A -85,B 0,C 180,E1 -6851.784,E2 -6851.784} C_VEL
LIN {X 0,Y 481.733,Z 346.48,A -85,B 0,C 180,E1 -6855.225,E2 -6855.225} C_VEL
LIN {X 0,Y 481.703,Z 346.479,A -85,B 0,C 180,E1 -6858.722,E2 -6858.722} C_VEL
LIN {X 0,Y 481.638,Z 346.493,A -85,B 0,C 180,E1 -6861.395,E2 -6861.395} C_VEL
LIN {X 0,Y 481.669,Z 346.482,A -85,B 0,C 180,E1 -6864.114,E2 -6864.114} C_VEL
LIN {X 0,Y 481.744,Z 346.479,A -85,B 0,C 180,E1 -6867.141,E2 -6867.141} C_VEL
LIN {X 0,Y 481.671,Z 346.484,A -85,B 0,C 180,E1 -6869.742,E2 -6869.742} C_VEL
LIN {X 0,Y 481.666,Z 346.485,A -85,B 0,C 180,E1 -6872.675,E2 -6872.675} C_VEL
LIN {X 0,Y 481.636,Z 346.488,A -85,B 0,C 180,E1 -6875.71,E2 -6875.71} C_VEL
LIN {X 0,Y 481.714,Z 346.481,A -85,B 0,C 180,E1 -6879.356,E2 -6879.356} C_VEL
LIN {X 0,Y 481.67,Z 346.482,A -85,B 0,C 180,E1 -6882.159,E2 -6882.159} C_VEL
LIN {X 0,Y 481.655,Z 346.486,A -85,B 0,C 180,E1 -6884.458,E2 -6884.458} C_VEL
LIN {X 0,Y 481.684,Z 346.485,A -85,B 0,C 180,E1 -6886.847,E2 -6886.847} C_VEL
LIN {X 0,Y 481.688,Z 346.48,A -85,B 0,C 180,E1 -6890.062,E2 -6890.062} C_VEL
LIN {X 0,Y 481.628,Z 346.492,A -85,B 0,C 180,E1 -6893.255,E2 -6893.255} C_VEL
LIN {X 0,Y 481.706,Z 346.48,A -85,B 0,C 180,E1 -6896.331,E2 -6896.331} C_VEL
LIN {X 0,Y 481.663,Z 346.488,A -85,B 0,C 180,E1 -6899.416,E2 -6899.416} C_VEL
LIN {X 0,Y 481.749,Z 346.586,A -85,B 0,C 180,E1 -6902.417,E2 -6902.417} C_VEL
LIN {X 0,Y 484.448,Z 359.917,A -85,B 0,C 180,E1 -6904.663,E2 -6904.663} C_VEL
LIN {X 0,Y 483.827,Z 375.968,A -85,B 0,C 180,E1 -6907.136,E2 -6907.136} C_VEL
LIN {X 0,Y 483.13,Z 394.858,A -85,B 0,C 180,E1 -6910.012,E2 -6910.012} C_VEL
LIN {X 0,Y 482.409,Z 416.467,A -85,B 0,C 180,E1 -6913.257,E2 -6913.257} C_VEL
LIN {X 0,Y 482.345,Z 418.089,A -85,B 0,C 180,E1 -6913.499,E2 -6913.499} C_VEL
LIN {X 0,Y 484.684,Z 436.549,A -85,B 0,C 180,E1 -6913.89,E2 -6913.89} C_VEL
LIN {X 0,Y 483.869,Z 527.682,A -85,B 0,C 180,E1 -6915.384,E2 -6915.384} C_VEL
LIN {X 0,Y 483.511,Z 541.278,A -85,B 0,C 180,E1 -6915.776,E2 -6915.776} C_VEL
LIN {X 0,Y 483.082,Z 554.184,A -85,B 0,C 180,E1 -6916.326,E2 -6916.326} C_VEL
LIN {X 0,Y 482.68,Z 566.8,A -85,B 0,C 180,E1 -6917.065,E2 -6917.065} C_VEL
LIN {X 0,Y 482.309,Z 577.666,A -85,B 0,C 180,E1 -6917.875,E2 -6917.875} C_VEL
LIN {X 0,Y 482.009,Z 587.253,A -85,B 0,C 180,E1 -6918.755,E2 -6918.755} C_VEL
LIN {X 0,Y 481.614,Z 595.798,A -85,B 0,C 180,E1 -6919.704,E2 -6919.704} C_VEL
LIN {X 0,Y 481.321,Z 605.065,A -85,B 0,C 180,E1 -6920.97,E2 -6920.97} C_VEL
LIN {X 0,Y 481.095,Z 612.525,A -85,B 0,C 180,E1 -6922.235,E2 -6922.235} C_VEL
LIN {X 0,Y 481.021,Z 618.398,A -85,B 0,C 180,E1 -6923.475,E2 -6923.475} C_VEL
LIN {X 0,Y 480.905,Z 623.838,A -85,B 0,C 180,E1 -6924.971,E2 -6924.971} C_VEL
LIN {X 0,Y 480.917,Z 626.205,A -85,B 0,C 180,E1 -6925.811,E2 -6925.811} C_VEL
LIN {X 0,Y 480.913,Z 628.128,A -85,B 0,C 180,E1 -6926.65,E2 -6926.65} C_VEL
LIN {X 0,Y 480.928,Z 629.575,A -85,B 0,C 180,E1 -6927.488,E2 -6927.488} C_VEL
LIN {X 0,Y 480.826,Z 630.581,A -85,B 0,C 180,E1 -6928.326,E2 -6928.326} C_VEL
LIN {X 0,Y 480.779,Z 631.188,A -85,B 0,C 180,E1 -6929.163,E2 -6929.163} C_VEL
LIN {X 0,Y 480.78,Z 631.39,A -85,B 0,C 180,E1 -6930.001,E2 -6930.001} C_VEL
LIN {X 0,Y 480.781,Z 631.138,A -85,B 0,C 180,E1 -6930.839,E2 -6930.839} C_VEL
LIN {X 0,Y 480.935,Z 629.415,A -85,B 0,C 180,E1 -6932.514,E2 -6932.514} C_VEL
LIN {X 0,Y 480.94,Z 627.918,A -85,B 0,C 180,E1 -6933.352,E2 -6933.352} C_VEL
LIN {X 0,Y 480.873,Z 624.793,A -85,B 0,C 180,E1 -6934.612,E2 -6934.612} C_VEL
LIN {X 0,Y 480.968,Z 620.584,A -85,B 0,C 180,E1 -6935.872,E2 -6935.872} C_VEL
LIN {X 0,Y 481.083,Z 615.158,A -85,B 0,C 180,E1 -6937.134,E2 -6937.134} C_VEL
LIN {X 0,Y 481.192,Z 608.326,A -85,B 0,C 180,E1 -6938.399,E2 -6938.399} C_VEL
LIN {X 0,Y 481.417,Z 599.833,A -85,B 0,C 180,E1 -6939.666,E2 -6939.666} C_VEL
LIN {X 0,Y 481.684,Z 591.151,A -85,B 0,C 180,E1 -6940.722,E2 -6940.722} C_VEL
LIN {X 0,Y 482.09,Z 580.451,A -85,B 0,C 180,E1 -6941.777,E2 -6941.777} C_VEL
LIN {X 0,Y 482.495,Z 568.405,A -85,B 0,C 180,E1 -6942.728,E2 -6942.728} C_VEL
LIN {X 0,Y 482.906,Z 556.354,A -85,B 0,C 180,E1 -6943.466,E2 -6943.466} C_VEL
LIN {X 0,Y 483.287,Z 543.892,A -85,B 0,C 180,E1 -6944.045,E2 -6944.045} C_VEL
LIN {X 0,Y 483.683,Z 531.291,A -85,B 0,C 180,E1 -6944.463,E2 -6944.463} C_VEL
LIN {X 0,Y 483.936,Z 517.085,A -85,B 0,C 180,E1 -6944.751,E2 -6944.751} C_VEL
LIN {X 0,Y 484.621,Z 435.371,A -85,B 0,C 180,E1 -6946.114,E2 -6946.114} C_VEL
LIN {X 0,Y 482.191,Z 415.736,A -85,B 0,C 180,E1 -6946.568,E2 -6946.568} C_VEL
LIN {X 0,Y 482.859,Z 394.268,A -85,B 0,C 180,E1 -6949.78,E2 -6949.78} C_VEL
LIN {X 0,Y 483.577,Z 374.018,A -85,B 0,C 180,E1 -6952.879,E2 -6952.879} C_VEL
LIN {X 0,Y 484.217,Z 359.81,A -85,B 0,C 180,E1 -6955.108,E2 -6955.108} C_VEL
LIN {X 0,Y 482.764,Z 351.214,A -85,B 0,C 180,E1 -6956.594,E2 -6956.594} C_VEL
LIN {X 0,Y 481.71,Z 346.485,A -85,B 0,C 180,E1 -6957.495,E2 -6957.495} C_VEL
LIN {X 0,Y 481.656,Z 346.489,A -85,B 0,C 180,E1 -6960.583,E2 -6960.583} C_VEL
LIN {X 0,Y 481.702,Z 346.483,A -85,B 0,C 180,E1 -6963.734,E2 -6963.734} C_VEL
LIN {X 0,Y 481.631,Z 346.493,A -85,B 0,C 180,E1 -6966.747,E2 -6966.747} C_VEL
LIN {X 0,Y 481.682,Z 346.483,A -85,B 0,C 180,E1 -6969.941,E2 -6969.941} C_VEL
LIN {X 0,Y 481.644,Z 346.49,A -85,B 0,C 180,E1 -6973.3,E2 -6973.3} C_VEL
LIN {X 0,Y 481.664,Z 346.485,A -85,B 0,C 180,E1 -6975.641,E2 -6975.641} C_VEL
LIN {X 0,Y 481.662,Z 346.49,A -85,B 0,C 180,E1 -6978.959,E2 -6978.959} C_VEL
LIN {X 0,Y 481.66,Z 346.485,A -85,B 0,C 180,E1 -6981.993,E2 -6981.993} C_VEL
LIN {X 0,Y 481.694,Z 346.483,A -85,B 0,C 180,E1 -6985.318,E2 -6985.318} C_VEL
LIN {X 0,Y 481.65,Z 346.488,A -85,B 0,C 180,E1 -6988.312,E2 -6988.312} C_VEL
LIN {X 0,Y 481.705,Z 346.483,A -85,B 0,C 180,E1 -6991.219,E2 -6991.219} C_VEL
LIN {X 0,Y 481.706,Z 346.481,A -85,B 0,C 180,E1 -6994.043,E2 -6994.043} C_VEL
LIN {X 0,Y 481.68,Z 346.488,A -85,B 0,C 180,E1 -6996.812,E2 -6996.812} C_VEL
LIN {X 0,Y 481.701,Z 346.483,A -85,B 0,C 180,E1 -6999.503,E2 -6999.503} C_VEL
LIN {X 0,Y 481.753,Z 346.622,A -85,B 0,C 180,E1 -7002.032,E2 -7002.032} C_VEL
LIN {X 0,Y 482.668,Z 352.436,A -85,B 0,C 180,E1 -7003.574,E2 -7003.574} C_VEL
LIN {X 0,Y 485.096,Z 361.849,A -85,B 0,C 180,E1 -7003.843,E2 -7003.843} C_VEL
LIN {X 0,Y 483.973,Z 458.882,A -85,B 0,C 180,E1 -7005.52,E2 -7005.52} C_VEL
LIN {X 0,Y 483.82,Z 471.918,A -85,B 0,C 180,E1 -7005.918,E2 -7005.918} C_VEL
LIN {X 0,Y 483.485,Z 483.927,A -85,B 0,C 180,E1 -7006.444,E2 -7006.444} C_VEL
LIN {X 0,Y 483.198,Z 495.895,A -85,B 0,C 180,E1 -7007.152,E2 -7007.152} C_VEL
LIN {X 0,Y 482.817,Z 507.48,A -85,B 0,C 180,E1 -7008.028,E2 -7008.028} C_VEL
LIN {X 0,Y 482.492,Z 516.461,A -85,B 0,C 180,E1 -7008.872,E2 -7008.872} C_VEL
LIN {X 0,Y 482.162,Z 525.654,A -85,B 0,C 180,E1 -7009.926,E2 -7009.926} C_VEL
LIN {X 0,Y 481.778,Z 534.563,A -85,B 0,C 180,E1 -7011.189,E2 -7011.189} C_VEL
LIN {X 0,Y 481.513,Z 541.696,A -85,B 0,C 180,E1 -7012.452,E2 -7012.452} C_VEL
LIN {X 0,Y 481.276,Z 547.343,A -85,B 0,C 180,E1 -7013.712,E2 -7013.712} C_VEL
LIN {X 0,Y 481.228,Z 551.752,A -85,B 0,C 180,E1 -7014.973,E2 -7014.973} C_VEL
LIN {X 0,Y 481.131,Z 554.073,A -85,B 0,C 180,E1 -7015.811,E2 -7015.811} C_VEL
LIN {X 0,Y 481.104,Z 555.958,A -85,B 0,C 180,E1 -7016.65,E2 -7016.65} C_VEL
LIN {X 0,Y 480.953,Z 557.405,A -85,B 0,C 180,E1 -7017.487,E2 -7017.487} C_VEL
LIN {X 0,Y 480.813,Z 559.008,A -85,B 0,C 180,E1 -7019.162,E2 -7019.162} C_VEL
LIN {X 0,Y 480.806,Z 559.219,A -85,B 0,C 180,E1 -7020,E2 -7020} C_VEL
LIN {X 0,Y 480.81,Z 558.996,A -85,B 0,C 180,E1 -7020.837,E2 -7020.837} C_VEL
LIN {X 0,Y 480.95,Z 557.327,A -85,B 0,C 180,E1 -7022.512,E2 -7022.512} C_VEL
LIN {X 0,Y 481.09,Z 555.889,A -85,B 0,C 180,E1 -7023.35,E2 -7023.35} C_VEL
LIN {X 0,Y 481.121,Z 552.899,A -85,B 0,C 180,E1 -7024.608,E2 -7024.608} C_VEL
LIN {X 0,Y 481.164,Z 548.855,A -85,B 0,C 180,E1 -7025.868,E2 -7025.868} C_VEL
LIN {X 0,Y 481.378,Z 542.713,A -85,B 0,C 180,E1 -7027.318,E2 -7027.318} C_VEL
LIN {X 0,Y 481.669,Z 535.792,A -85,B 0,C 180,E1 -7028.601,E2 -7028.601} C_VEL
LIN {X 0,Y 481.978,Z 527.303,A -85,B 0,C 180,E1 -7029.865,E2 -7029.865} C_VEL
LIN {X 0,Y 482.287,Z 518.538,A -85,B 0,C 180,E1 -7030.92,E2 -7030.92} C_VEL
LIN {X 0,Y 482.759,Z 507.734,A -85,B 0,C 180,E1 -7031.973,E2 -7031.973} C_VEL
LIN {X 0,Y 483.1,Z 496.641,A -85,B 0,C 180,E1 -7032.838,E2 -7032.838} C_VEL
LIN {X 0,Y 483.412,Z 484.845,A -85,B 0,C 180,E1 -7033.558,E2 -7033.558} C_VEL
LIN {X 0,Y 483.794,Z 472.261,A -85,B 0,C 180,E1 -7034.136,E2 -7034.136} C_VEL
LIN {X 0,Y 484.009,Z 460.063,A -85,B 0,C 180,E1 -7034.533,E2 -7034.533} C_VEL
LIN {X 0,Y 484.107,Z 443.447,A -85,B 0,C 180,E1 -7034.852,E2 -7034.852} C_VEL
LIN {X 0,Y 484.821,Z 361.146,A -85,B 0,C 180,E1 -7036.192,E2 -7036.192} C_VEL
LIN {X 0,Y 482.144,Z 349.395,A -85,B 0,C 180,E1 -7036.499,E2 -7036.499} C_VEL
LIN {X 0,Y 481.729,Z 346.483,A -85,B 0,C 180,E1 -7037.238,E2 -7037.238} C_VEL
LIN {X 0,Y 481.7,Z 346.48,A -85,B 0,C 180,E1 -7040.497,E2 -7040.497} C_VEL
LIN {X 0,Y 481.67,Z 346.488,A -85,B 0,C 180,E1 -7043.201,E2 -7043.201} C_VEL
LIN {X 0,Y 481.701,Z 346.481,A -85,B 0,C 180,E1 -7045.957,E2 -7045.957} C_VEL
LIN {X 0,Y 481.705,Z 346.482,A -85,B 0,C 180,E1 -7048.781,E2 -7048.781} C_VEL
LIN {X 0,Y 481.661,Z 346.485,A -85,B 0,C 180,E1 -7052.189,E2 -7052.189} C_VEL
LIN {X 0,Y 481.693,Z 346.483,A -85,B 0,C 180,E1 -7054.682,E2 -7054.682} C_VEL
LIN {X 0,Y 481.659,Z 346.485,A -85,B 0,C 180,E1 -7058.007,E2 -7058.007} C_VEL
LIN {X 0,Y 481.661,Z 346.489,A -85,B 0,C 180,E1 -7061.041,E2 -7061.041} C_VEL
LIN {X 0,Y 481.664,Z 346.486,A -85,B 0,C 180,E1 -7064.457,E2 -7064.457} C_VEL
LIN {X 0,Y 481.652,Z 346.486,A -85,B 0,C 180,E1 -7067.839,E2 -7067.839} C_VEL
LIN {X 0,Y 481.685,Z 346.486,A -85,B 0,C 180,E1 -7070.651,E2 -7070.651} C_VEL
LIN {X 0,Y 481.613,Z 346.491,A -85,B 0,C 180,E1 -7072.858,E2 -7072.858} C_VEL
LIN {X 0,Y 480.962,Z 346.576,A -85,B 0,C 180,E1 -7073.555,E2 -7073.555} C_VEL
LIN {X 0,Y 478.124,Z 346.931,A -85,B 0,C 180,E1 -7074.689,E2 -7074.689} C_VEL
LIN {X 0,Y 475.727,Z 347.225,A -85,B 0,C 180,E1 -7075.602,E2 -7075.602} C_VEL
LIN {X 0,Y 474.711,Z 347.352,A -85,B 0,C 180,E1 -7076.308,E2 -7076.308} C_VEL
LIN {X 0,Y 474.636,Z 347.362,A -85,B 0,C 180,E1 -7076.547,E2 -7076.547} C_VEL
LIN {X 0,Y 474.609,Z 347.363,A -85,B 0,C 180,E1 -7079.769,E2 -7079.769} C_VEL
LIN {X 0,Y 474.701,Z 347.357,A -85,B 0,C 180,E1 -7082.679,E2 -7082.679} C_VEL
LIN {X 0,Y 474.663,Z 347.357,A -85,B 0,C 180,E1 -7085.507,E2 -7085.507} C_VEL
LIN {X 0,Y 474.674,Z 347.358,A -85,B 0,C 180,E1 -7089.185,E2 -7089.185} C_VEL
LIN {X 0,Y 474.661,Z 347.357,A -85,B 0,C 180,E1 -7091.884,E2 -7091.884} C_VEL
LIN {X 0,Y 474.704,Z 347.357,A -85,B 0,C 180,E1 -7094.544,E2 -7094.544} C_VEL
LIN {X 0,Y 474.708,Z 347.352,A -85,B 0,C 180,E1 -7098.037,E2 -7098.037} C_VEL
LIN {X 0,Y 474.731,Z 347.348,A -85,B 0,C 180,E1 -7101.486,E2 -7101.486} C_VEL
LIN {X 0,Y 474.774,Z 347.344,A -85,B 0,C 180,E1 -7104.051,E2 -7104.051} C_VEL
LIN {X 0,Y 474.897,Z 347.327,A -85,B 0,C 180,E1 -7107.454,E2 -7107.454} C_VEL
LIN {X 0,Y 474.914,Z 347.327,A -85,B 0,C 180,E1 -7109.999,E2 -7109.999} C_VEL
LIN {X 0,Y 474.897,Z 347.331,A -85,B 0,C 180,E1 -7112.544,E2 -7112.544} C_VEL
LIN {X 0,Y 474.783,Z 347.343,A -85,B 0,C 180,E1 -7115.947,E2 -7115.947} C_VEL
LIN {X 0,Y 474.729,Z 347.352,A -85,B 0,C 180,E1 -7118.512,E2 -7118.512} C_VEL
LIN {X 0,Y 474.705,Z 347.354,A -85,B 0,C 180,E1 -7121.961,E2 -7121.961} C_VEL
LIN {X 0,Y 474.701,Z 347.353,A -85,B 0,C 180,E1 -7125.776,E2 -7125.776} C_VEL
LIN {X 0,Y 474.665,Z 347.357,A -85,B 0,C 180,E1 -7129.009,E2 -7129.009} C_VEL
LIN {X 0,Y 474.589,Z 347.367,A -85,B 0,C 180,E1 -7131.728,E2 -7131.728} C_VEL
LIN {X 0,Y 474.657,Z 347.36,A -85,B 0,C 180,E1 -7134.492,E2 -7134.492} C_VEL
LIN {X 0,Y 474.696,Z 347.352,A -85,B 0,C 180,E1 -7137.338,E2 -7137.338} C_VEL
LIN {X 0,Y 474.607,Z 347.364,A -85,B 0,C 180,E1 -7140.81,E2 -7140.81} C_VEL
LIN {X 0,Y 474.634,Z 347.365,A -85,B 0,C 180,E1 -7143.983,E2 -7143.983} C_VEL
LIN {X 0,Y 474.572,Z 347.367,A -85,B 0,C 180,E1 -7146.899,E2 -7146.899} C_VEL
LIN {X 0,Y 474.661,Z 347.359,A -85,B 0,C 180,E1 -7149.652,E2 -7149.652} C_VEL
LIN {X 0,Y 474.645,Z 347.358,A -85,B 0,C 180,E1 -7152.929,E2 -7152.929} C_VEL
LIN {X 0,Y 474.612,Z 347.369,A -85,B 0,C 180,E1 -7155.895,E2 -7155.895} C_VEL
LIN {X 0,Y 474.641,Z 347.358,A -85,B 0,C 180,E1 -7159.037,E2 -7159.037} C_VEL
LIN {X 0,Y 474.612,Z 347.366,A -85,B 0,C 180,E1 -7161.702,E2 -7161.702} C_VEL
LIN {X 0,Y 474.622,Z 347.361,A -85,B 0,C 180,E1 -7164.725,E2 -7164.725} C_VEL
LIN {X 0,Y 474.63,Z 347.366,A -85,B 0,C 180,E1 -7167.787,E2 -7167.787} C_VEL
LIN {X 0,Y 474.623,Z 347.36,A -85,B 0,C 180,E1 -7170.882,E2 -7170.882} C_VEL
LIN {X 0,Y 474.658,Z 347.361,A -85,B 0,C 180,E1 -7173.628,E2 -7173.628} C_VEL
LIN {X 0,Y 474.626,Z 347.36,A -85,B 0,C 180,E1 -7176.641,E2 -7176.641} C_VEL
LIN {X 0,Y 474.647,Z 347.36,A -85,B 0,C 180,E1 -7180.089,E2 -7180.089} C_VEL
LIN {X 0,Y 474.642,Z 347.357,A -85,B 0,C 180,E1 -7182.774,E2 -7182.774} C_VEL
LIN {X 0,Y 474.639,Z 347.362,A -85,B 0,C 180,E1 -7185.421,E2 -7185.421} C_VEL
LIN {X 0,Y 474.73,Z 347.349,A -85,B 0,C 180,E1 -7188.038,E2 -7188.038} C_VEL
LIN {X 0,Y 474.72,Z 347.354,A -85,B 0,C 180,E1 -7191.486,E2 -7191.486} C_VEL
LIN {X 0,Y 474.77,Z 347.343,A -85,B 0,C 180,E1 -7194.052,E2 -7194.052} C_VEL
LIN {X 0,Y 474.886,Z 347.334,A -85,B 0,C 180,E1 -7197.455,E2 -7197.455} C_VEL
LIN {X 0,Y 474.867,Z 347.33,A -85,B 0,C 180,E1 -7200.848,E2 -7200.848} C_VEL
LIN {X 0,Y 474.886,Z 347.326,A -85,B 0,C 180,E1 -7202.545,E2 -7202.545} C_VEL
LIN {X 0,Y 474.78,Z 347.342,A -85,B 0,C 180,E1 -7205.948,E2 -7205.948} C_VEL
LIN {X 0,Y 474.719,Z 347.347,A -85,B 0,C 180,E1 -7208.514,E2 -7208.514} C_VEL
LIN {X 0,Y 474.73,Z 347.348,A -85,B 0,C 180,E1 -7211.962,E2 -7211.962} C_VEL
LIN {X 0,Y 474.671,Z 347.356,A -85,B 0,C 180,E1 -7215.769,E2 -7215.769} C_VEL
LIN {X 0,Y 474.656,Z 347.359,A -85,B 0,C 180,E1 -7219.011,E2 -7219.011} C_VEL
LIN {X 0,Y 474.582,Z 347.367,A -85,B 0,C 180,E1 -7221.729,E2 -7221.729} C_VEL
LIN {X 0,Y 474.651,Z 347.357,A -85,B 0,C 180,E1 -7224.493,E2 -7224.493} C_VEL
LIN {X 0,Y 474.69,Z 347.358,A -85,B 0,C 180,E1 -7227.339,E2 -7227.339} C_VEL
LIN {X 0,Y 474.597,Z 347.366,A -85,B 0,C 180,E1 -7230.811,E2 -7230.811} C_VEL
LIN {X 0,Y 474.631,Z 347.359,A -85,B 0,C 180,E1 -7233.985,E2 -7233.985} C_VEL
LIN {X 0,Y 474.571,Z 347.371,A -85,B 0,C 180,E1 -7236.901,E2 -7236.901} C_VEL
LIN {X 0,Y 474.649,Z 347.358,A -85,B 0,C 180,E1 -7239.653,E2 -7239.653} C_VEL
LIN {X 0,Y 474.647,Z 347.362,A -85,B 0,C 180,E1 -7242.931,E2 -7242.931} C_VEL
LIN {X 0,Y 474.613,Z 347.362,A -85,B 0,C 180,E1 -7245.897,E2 -7245.897} C_VEL
LIN {X 0,Y 474.64,Z 347.365,A -85,B 0,C 180,E1 -7249.039,E2 -7249.039} C_VEL
LIN {X 0,Y 474.616,Z 347.362,A -85,B 0,C 180,E1 -7251.703,E2 -7251.703} C_VEL
LIN {X 0,Y 474.627,Z 347.364,A -85,B 0,C 180,E1 -7254.727,E2 -7254.727} C_VEL
LIN {X 0,Y 474.635,Z 347.359,A -85,B 0,C 180,E1 -7257.789,E2 -7257.789} C_VEL
LIN {X 0,Y 474.631,Z 347.368,A -85,B 0,C 180,E1 -7260.884,E2 -7260.884} C_VEL
LIN {X 0,Y 474.678,Z 347.438,A -85,B 0,C 180,E1 -7262.199,E2 -7262.199} C_VEL
LIN {X 0,Y 477.488,Z 361.138,A -85,B 0,C 180,E1 -7264.542,E2 -7264.542} C_VEL
LIN {X 0,Y 477.027,Z 374.005,A -85,B 0,C 180,E1 -7266.561,E2 -7266.561} C_VEL
LIN {X 0,Y 476.228,Z 392.928,A -85,B 0,C 180,E1 -7269.484,E2 -7269.484} C_VEL
LIN {X 0,Y 475.447,Z 414.688,A -85,B 0,C 180,E1 -7272.805,E2 -7272.805} C_VEL
LIN {X 0,Y 475.377,Z 417.733,A -85,B 0,C 180,E1 -7273.262,E2 -7273.262} C_VEL
LIN {X 0,Y 477.841,Z 437.345,A -85,B 0,C 180,E1 -7273.683,E2 -7273.683} C_VEL
LIN {X 0,Y 476.959,Z 527.323,A -85,B 0,C 180,E1 -7275.194,E2 -7275.194} C_VEL
LIN {X 0,Y 476.593,Z 540.844,A -85,B 0,C 180,E1 -7275.592,E2 -7275.592} C_VEL
LIN {X 0,Y 476.18,Z 553.208,A -85,B 0,C 180,E1 -7276.124,E2 -7276.124} C_VEL
LIN {X 0,Y 475.781,Z 564.338,A -85,B 0,C 180,E1 -7276.765,E2 -7276.765} C_VEL
LIN {X 0,Y 475.321,Z 576.181,A -85,B 0,C 180,E1 -7277.638,E2 -7277.638} C_VEL
LIN {X 0,Y 474.982,Z 586.503,A -85,B 0,C 180,E1 -7278.587,E2 -7278.587} C_VEL
LIN {X 0,Y 474.577,Z 595.1,A -85,B 0,C 180,E1 -7279.549,E2 -7279.549} C_VEL
LIN {X 0,Y 474.255,Z 604.418,A -85,B 0,C 180,E1 -7280.835,E2 -7280.835} C_VEL
LIN {X 0,Y 474.034,Z 611.914,A -85,B 0,C 180,E1 -7282.119,E2 -7282.119} C_VEL
LIN {X 0,Y 473.937,Z 618.277,A -85,B 0,C 180,E1 -7283.487,E2 -7283.487} C_VEL
LIN {X 0,Y 473.842,Z 623.285,A -85,B 0,C 180,E1 -7284.895,E2 -7284.895} C_VEL
LIN {X 0,Y 473.815,Z 625.657,A -85,B 0,C 180,E1 -7285.748,E2 -7285.748} C_VEL
LIN {X 0,Y 473.841,Z 627.589,A -85,B 0,C 180,E1 -7286.6,E2 -7286.6} C_VEL
LIN {X 0,Y 473.867,Z 629.045,A -85,B 0,C 180,E1 -7287.451,E2 -7287.451} C_VEL
LIN {X 0,Y 473.761,Z 630.054,A -85,B 0,C 180,E1 -7288.301,E2 -7288.301} C_VEL
LIN {X 0,Y 473.707,Z 630.659,A -85,B 0,C 180,E1 -7289.151,E2 -7289.151} C_VEL
LIN {X 0,Y 473.704,Z 630.86,A -85,B 0,C 180,E1 -7290.001,E2 -7290.001} C_VEL
LIN {X 0,Y 473.709,Z 630.605,A -85,B 0,C 180,E1 -7290.851,E2 -7290.851} C_VEL
LIN {X 0,Y 473.762,Z 629.939,A -85,B 0,C 180,E1 -7291.701,E2 -7291.701} C_VEL
LIN {X 0,Y 473.875,Z 628.868,A -85,B 0,C 180,E1 -7292.551,E2 -7292.551} C_VEL
LIN {X 0,Y 473.854,Z 626.408,A -85,B 0,C 180,E1 -7293.828,E2 -7293.828} C_VEL
LIN {X 0,Y 473.844,Z 622.907,A -85,B 0,C 180,E1 -7295.107,E2 -7295.107} C_VEL
LIN {X 0,Y 473.95,Z 617.719,A -85,B 0,C 180,E1 -7296.528,E2 -7296.528} C_VEL
LIN {X 0,Y 474.037,Z 611.276,A -85,B 0,C 180,E1 -7297.883,E2 -7297.883} C_VEL
LIN {X 0,Y 474.246,Z 603.628,A -85,B 0,C 180,E1 -7299.168,E2 -7299.168} C_VEL
LIN {X 0,Y 474.535,Z 594.122,A -85,B 0,C 180,E1 -7300.454,E2 -7300.454} C_VEL
LIN {X 0,Y 474.821,Z 584.232,A -85,B 0,C 180,E1 -7301.527,E2 -7301.527} C_VEL
LIN {X 0,Y 475.267,Z 574.103,A -85,B 0,C 180,E1 -7302.426,E2 -7302.426} C_VEL
LIN {X 0,Y 475.724,Z 562.786,A -85,B 0,C 180,E1 -7303.238,E2 -7303.238} C_VEL
LIN {X 0,Y 476.14,Z 550.265,A -85,B 0,C 180,E1 -7303.933,E2 -7303.933} C_VEL
LIN {X 0,Y 476.573,Z 536.485,A -85,B 0,C 180,E1 -7304.492,E2 -7304.492} C_VEL
LIN {X 0,Y 476.974,Z 523.542,A -85,B 0,C 180,E1 -7304.835,E2 -7304.835} C_VEL
LIN {X 0,Y 477.779,Z 435.765,A -85,B 0,C 180,E1 -7306.351,E2 -7306.351} C_VEL
LIN {X 0,Y 475.187,Z 415.045,A -85,B 0,C 180,E1 -7306.848,E2 -7306.848} C_VEL
LIN {X 0,Y 475.908,Z 393.839,A -85,B 0,C 180,E1 -7310.082,E2 -7310.082} C_VEL
LIN {X 0,Y 476.647,Z 375.168,A -85,B 0,C 180,E1 -7313.001,E2 -7313.001} C_VEL
LIN {X 0,Y 477.333,Z 360.985,A -85,B 0,C 180,E1 -7315.277,E2 -7315.277} C_VEL
LIN {X 0,Y 475.547,Z 351.181,A -85,B 0,C 180,E1 -7317.03,E2 -7317.03} C_VEL
LIN {X 0,Y 474.663,Z 347.363,A -85,B 0,C 180,E1 -7317.768,E2 -7317.768} C_VEL
LIN {X 0,Y 474.61,Z 347.369,A -85,B 0,C 180,E1 -7320.811,E2 -7320.811} C_VEL
LIN {X 0,Y 474.643,Z 347.362,A -85,B 0,C 180,E1 -7323.984,E2 -7323.984} C_VEL
LIN {X 0,Y 474.578,Z 347.373,A -85,B 0,C 180,E1 -7326.9,E2 -7326.9} C_VEL
LIN {X 0,Y 474.633,Z 347.363,A -85,B 0,C 180,E1 -7329.648,E2 -7329.648} C_VEL
LIN {X 0,Y 474.62,Z 347.367,A -85,B 0,C 180,E1 -7332.935,E2 -7332.935} C_VEL
LIN {X 0,Y 474.615,Z 347.363,A -85,B 0,C 180,E1 -7335.895,E2 -7335.895} C_VEL
LIN {X 0,Y 474.633,Z 347.365,A -85,B 0,C 180,E1 -7339.041,E2 -7339.041} C_VEL
LIN {X 0,Y 474.615,Z 347.363,A -85,B 0,C 180,E1 -7341.704,E2 -7341.704} C_VEL
LIN {X 0,Y 474.629,Z 347.364,A -85,B 0,C 180,E1 -7344.726,E2 -7344.726} C_VEL
LIN {X 0,Y 474.641,Z 347.36,A -85,B 0,C 180,E1 -7347.788,E2 -7347.788} C_VEL
LIN {X 0,Y 474.63,Z 347.366,A -85,B 0,C 180,E1 -7350.885,E2 -7350.885} C_VEL
LIN {X 0,Y 474.666,Z 347.358,A -85,B 0,C 180,E1 -7353.629,E2 -7353.629} C_VEL
LIN {X 0,Y 474.641,Z 347.365,A -85,B 0,C 180,E1 -7356.641,E2 -7356.641} C_VEL
LIN {X 0,Y 474.659,Z 347.361,A -85,B 0,C 180,E1 -7360.09,E2 -7360.09} C_VEL
LIN {X 0,Y 474.721,Z 347.526,A -85,B 0,C 180,E1 -7361.759,E2 -7361.759} C_VEL
LIN {X 0,Y 475.708,Z 353.353,A -85,B 0,C 180,E1 -7363.296,E2 -7363.296} C_VEL
LIN {X 0,Y 478.317,Z 362.706,A -85,B 0,C 180,E1 -7363.585,E2 -7363.585} C_VEL
LIN {X 0,Y 477.128,Z 459.332,A -85,B 0,C 180,E1 -7365.308,E2 -7365.308} C_VEL
LIN {X 0,Y 476.954,Z 472.356,A -85,B 0,C 180,E1 -7365.711,E2 -7365.711} C_VEL
LIN {X 0,Y 476.603,Z 484.394,A -85,B 0,C 180,E1 -7366.244,E2 -7366.244} C_VEL
LIN {X 0,Y 476.304,Z 496.366,A -85,B 0,C 180,E1 -7366.963,E2 -7366.963} C_VEL
LIN {X 0,Y 475.897,Z 507.97,A -85,B 0,C 180,E1 -7367.852,E2 -7367.852} C_VEL
LIN {X 0,Y 475.549,Z 516.975,A -85,B 0,C 180,E1 -7368.707,E2 -7368.707} C_VEL
LIN {X 0,Y 475.197,Z 526.18,A -85,B 0,C 180,E1 -7369.777,E2 -7369.777} C_VEL
LIN {X 0,Y 474.797,Z 535.093,A -85,B 0,C 180,E1 -7371.059,E2 -7371.059} C_VEL
LIN {X 0,Y 474.485,Z 542.236,A -85,B 0,C 180,E1 -7372.339,E2 -7372.339} C_VEL
LIN {X 0,Y 474.213,Z 548.367,A -85,B 0,C 180,E1 -7373.745,E2 -7373.745} C_VEL
LIN {X 0,Y 474.117,Z 553.542,A -85,B 0,C 180,E1 -7375.323,E2 -7375.323} C_VEL
LIN {X 0,Y 474.056,Z 556.514,A -85,B 0,C 180,E1 -7376.6,E2 -7376.6} C_VEL
LIN {X 0,Y 473.898,Z 557.959,A -85,B 0,C 180,E1 -7377.45,E2 -7377.45} C_VEL
LIN {X 0,Y 473.738,Z 559.555,A -85,B 0,C 180,E1 -7379.15,E2 -7379.15} C_VEL
LIN {X 0,Y 473.729,Z 559.759,A -85,B 0,C 180,E1 -7380,E2 -7380} C_VEL
LIN {X 0,Y 473.736,Z 559.524,A -85,B 0,C 180,E1 -7380.85,E2 -7380.85} C_VEL
LIN {X 0,Y 473.894,Z 557.833,A -85,B 0,C 180,E1 -7382.55,E2 -7382.55} C_VEL
LIN {X 0,Y 474.04,Z 556.379,A -85,B 0,C 180,E1 -7383.4,E2 -7383.4} C_VEL
LIN {X 0,Y 474.071,Z 553.364,A -85,B 0,C 180,E1 -7384.677,E2 -7384.677} C_VEL
LIN {X 0,Y 474.124,Z 549.289,A -85,B 0,C 180,E1 -7385.956,E2 -7385.956} C_VEL
LIN {X 0,Y 474.327,Z 544.222,A -85,B 0,C 180,E1 -7387.192,E2 -7387.192} C_VEL
LIN {X 0,Y 474.592,Z 537.384,A -85,B 0,C 180,E1 -7388.516,E2 -7388.516} C_VEL
LIN {X 0,Y 474.9,Z 529.13,A -85,B 0,C 180,E1 -7389.799,E2 -7389.799} C_VEL
LIN {X 0,Y 475.259,Z 520.676,A -85,B 0,C 180,E1 -7390.868,E2 -7390.868} C_VEL
LIN {X 0,Y 475.696,Z 510.234,A -85,B 0,C 180,E1 -7391.937,E2 -7391.937} C_VEL
LIN {X 0,Y 476.131,Z 498.457,A -85,B 0,C 180,E1 -7392.9,E2 -7392.9} C_VEL
LIN {X 0,Y 476.45,Z 486.694,A -85,B 0,C 180,E1 -7393.651,E2 -7393.651} C_VEL
LIN {X 0,Y 476.79,Z 474.524,A -85,B 0,C 180,E1 -7394.24,E2 -7394.24} C_VEL
LIN {X 0,Y 477.054,Z 461.354,A -85,B 0,C 180,E1 -7394.695,E2 -7394.695} C_VEL
LIN {X 0,Y 477.203,Z 447.073,A -85,B 0,C 180,E1 -7394.99,E2 -7394.99} C_VEL
LIN {X 0,Y 478.053,Z 362.249,A -85,B 0,C 180,E1 -7396.402,E2 -7396.402} C_VEL
LIN {X 0,Y 475.103,Z 349.822,A -85,B 0,C 180,E1 -7396.737,E2 -7396.737} C_VEL
LIN {X 0,Y 474.686,Z 347.36,A -85,B 0,C 180,E1 -7397.335,E2 -7397.335} C_VEL
LIN {X 0,Y 474.659,Z 347.359,A -85,B 0,C 180,E1 -7399.91,E2 -7399.91} C_VEL
LIN {X 0,Y 474.64,Z 347.363,A -85,B 0,C 180,E1 -7403.358,E2 -7403.358} C_VEL
LIN {X 0,Y 474.662,Z 347.357,A -85,B 0,C 180,E1 -7406.371,E2 -7406.371} C_VEL
LIN {X 0,Y 474.626,Z 347.365,A -85,B 0,C 180,E1 -7409.252,E2 -7409.252} C_VEL
LIN {X 0,Y 474.619,Z 347.363,A -85,B 0,C 180,E1 -7412.43,E2 -7412.43} C_VEL
LIN {X 0,Y 474.619,Z 347.366,A -85,B 0,C 180,E1 -7415.469,E2 -7415.469} C_VEL
LIN {X 0,Y 474.616,Z 347.364,A -85,B 0,C 180,E1 -7418.457,E2 -7418.457} C_VEL
LIN {X 0,Y 474.632,Z 347.364,A -85,B 0,C 180,E1 -7420.959,E2 -7420.959} C_VEL
LIN {X 0,Y 474.614,Z 347.363,A -85,B 0,C 180,E1 -7424.104,E2 -7424.104} C_VEL
LIN {X 0,Y 474.619,Z 347.365,A -85,B 0,C 180,E1 -7427.065,E2 -7427.065} C_VEL
LIN {X 0,Y 474.649,Z 347.36,A -85,B 0,C 180,E1 -7430.454,E2 -7430.454} C_VEL
LIN {X 0,Y 474.593,Z 347.366,A -85,B 0,C 180,E1 -7433.676,E2 -7433.676} C_VEL
LIN {X 0,Y 474.636,Z 347.362,A -85,B 0,C 180,E1 -7436.547,E2 -7436.547} C_VEL
LIN {X 0,Y 473.983,Z 347.447,A -85,B 0,C 180,E1 -7437.255,E2 -7437.255} C_VEL
LIN {X 0,Y 471.11,Z 347.803,A -85,B 0,C 180,E1 -7438.406,E2 -7438.406} C_VEL
LIN {X 0,Y 468.675,Z 348.105,A -85,B 0,C 180,E1 -7439.333,E2 -7439.333} C_VEL
LIN {X 0,Y 467.638,Z 348.233,A -85,B 0,C 180,E1 -7440.05,E2 -7440.05} C_VEL
